    |   movel(pose_trans(ref_frame,p[0.022855, 0.074672, -0.000125, 0.000000, 3.141593, 0.000000]),accel_mss,speed_ms,0,0.001)
    |   movel(pose_trans(ref_frame,p[0.022965, 0.074913, -0.000125, -0.000000, 3.141593, -0.000000]),accel_mss,speed_ms,0,0.001)
    |   movel(pose_trans(ref_frame,p[0.022969, 0.075189, -0.000125, 0.000000, 3.141593, -0.000000]),accel_mss,speed_ms,0,0.001)
    |   movel(pose_trans(ref_frame,p[0.022613, 0.076078, -0.000125, -0.000000, 3.141593, 0.000000]),accel_mss,speed_ms,0,0.001)
    |   movel(pose_trans(ref_frame,p[0.022075, 0.076866, -0.000125, 0.000000, 3.141593, 0.000000]),accel_mss,speed_ms,0,0.001)
    |   movel(pose_trans(ref_frame,p[0.021271, 0.078122, -0.000125, 0.000000, 3.141593, -0.000000]),accel_mss,speed_ms,0,0.001)
    |   movel(pose_trans(ref_frame,p[0.022029, 0.079079, -0.000125, 0.000000, 3.141593, 0.000000]),accel_mss,speed_ms,0,0.001)
    |   movel(pose_trans(ref_frame,p[0.021683, 0.080650, -0.000125, -0.000000, 3.141593, 0.000000]),accel_mss,speed_ms,0,0.001)
    |   movel(pose_trans(ref_frame,p[0.020753, 0.081998, -0.000125, -0.000000, 3.141593, 0.000000]),accel_mss,speed_ms,0,0.001)
    |   movel(pose_trans(ref_frame,p[0.019633, 0.083228, -0.000125, -0.000000, 3.141593, -0.000000]),accel_mss,speed_ms,0,0.001)
    |   movel(pose_trans(ref_frame,p[0.018817, 0.084642, -0.000125, -0.000000, 3.141593, 0.000000]),accel_mss,speed_ms,0,0.001)
    |   movel(pose_trans(ref_frame,p[0.018857, 0.085057, -0.000125, -0.000000, 3.141593, 0.000000]),accel_mss,speed_ms,0,0.001)
    |   movel(pose_trans(ref_frame,p[0.019145, 0.085240, -0.000125, -0.000000, 3.141593, -0.000000]),accel_mss,speed_ms,0,0.001)
    |   movel(pose_trans(ref_frame,p[0.019287, 0.085189, -0.000125, -0.000000, 3.141593, 0.000000]),accel_mss,speed_ms,0,0.001)
    |   movel(pose_trans(ref_frame,p[0.019408, 0.085093, -0.000125, -0.000000, 3.141593, -0.000000]),accel_mss,speed_ms,0,0.001)
    |   movel(pose_trans(ref_frame,p[0.020443, 0.084055, -0.000125, 0.000000, 3.141593, 0.000000]),accel_mss,speed_ms,0,0.001)
    |   movel(pose_trans(ref_frame,p[0.021348, 0.082902, -0.000125, -0.000000, 3.141593, -0.000000]),accel_mss,speed_ms,0,0.001)
    |   movel(pose_trans(ref_frame,p[0.021279, 0.084884, -0.000125, -0.000000, 3.141593, -0.000000]),accel_mss,speed_ms,0,0.001)
    |   movel(pose_trans(ref_frame,p[0.019878, 0.086502, -0.000125, 0.000000, 3.141593, 0.000000]),accel_mss,speed_ms,0,0.001)
    |   movel(pose_trans(ref_frame,p[0.019692, 0.086795, -0.000125, 0.000000, 3.141593, -0.000000]),accel_mss,speed_ms,0,0.001)
    |   movel(pose_trans(ref_frame,p[0.019677, 0.087111, -0.000125, 0.000000, 3.141593, -0.000000]),accel_mss,speed_ms,0,0.001)
    |   movel(pose_trans(ref_frame,p[0.020252, 0.087228, -0.000125, -0.000000, 3.141593, 0.000000]),accel_mss,speed_ms,0,0.001)
    |   movel(pose_trans(ref_frame,p[0.020628, 0.087249, -0.000125, -0.000000, 3.141593, 0.000000]),accel_mss,speed_ms,0,0.001)
    |   movel(pose_trans(ref_frame,p[0.020630, 0.087969, -0.000125, -0.000000, 3.141593, -0.000000]),accel_mss,speed_ms,0,0.001)
    |   movel(pose_trans(ref_frame,p[0.020204, 0.088627, -0.000125, -0.000000, 3.141593, 0.000000]),accel_mss,speed_ms,0,0.001)
    |   movel(pose_trans(ref_frame,p[0.019352, 0.090039, -0.000125, 0.000000, 3.141593, -0.000000]),accel_mss,speed_ms,0,0.001)
    |   movel(pose_trans(ref_frame,p[0.018472, 0.091435, -0.000125, -0.000000, 3.141593, 0.000000]),accel_mss,speed_ms,0,0.001)
    |   movel(pose_trans(ref_frame,p[0.018239, 0.092061, -0.000125, 0.000000, 3.141593, 0.000000]),accel_mss,speed_ms,0,0.001)
    |   movel(pose_trans(ref_frame,p[0.018456, 0.092576, -0.000125, -0.000000, 3.141593, 0.000000]),accel_mss,speed_ms,0,0.001)
    |   movel(pose_trans(ref_frame,p[0.018989, 0.092581, -0.000125, 0.000000, 3.141593, -0.000000]),accel_mss,speed_ms,0,0.001)
    |   movel(pose_trans(ref_frame,p[0.019468, 0.092180, -0.000125, 0.000000, 3.141593, -0.000000]),accel_mss,speed_ms,0,0.001)
    |   movel(pose_trans(ref_frame,p[0.021768, 0.089335, -0.000125, -0.000000, 3.141593, -0.000000]),accel_mss,speed_ms,0,0.001)
    |   movel(pose_trans(ref_frame,p[0.023782, 0.086280, -0.000125, 0.000000, 3.141593, 0.000000]),accel_mss,speed_ms,0,0.001)
    |   movel(pose_trans(ref_frame,p[0.024110, 0.085688, -0.000125, 0.000000, 3.141593, 0.000000]),accel_mss,speed_ms,0,0.001)
    |   movel(pose_trans(ref_frame,p[0.024349, 0.085059, -0.000125, -0.000000, 3.141593, -0.000000]),accel_mss,speed_ms,0,0.001)
    |   movel(pose_trans(ref_frame,p[0.024445, 0.084271, -0.000125, 0.000000, 3.141593, 0.000000]),accel_mss,speed_ms,0,0.001)
    |   movel(pose_trans(ref_frame,p[0.024416, 0.083472, -0.000125, 0.000000, 3.141593, -0.000000]),accel_mss,speed_ms,0,0.001)
    |   movel(pose_trans(ref_frame,p[0.023805, 0.080672, -0.000125, -0.000000, 3.141593, -0.000000]),accel_mss,speed_ms,0,0.001)
    |   movel(pose_trans(ref_frame,p[0.024617, 0.078088, -0.000125, 0.000000, 3.141593, -0.000000]),accel_mss,speed_ms,0,0.001)
    |   movel(pose_trans(ref_frame,p[0.025018, 0.077876, -0.000125, 0.000000, 3.141593, 0.000000]),accel_mss,speed_ms,0,0.001)
    |   movel(pose_trans(ref_frame,p[0.025324, 0.077583, -0.000125, -0.000000, 3.141593, -0.000000]),accel_mss,speed_ms,0,0.001)
    |   movel(pose_trans(ref_frame,p[0.025361, 0.077273, -0.000125, 0.000000, 3.141593, 0.000000]),accel_mss,speed_ms,0,0.001)
    |   movel(pose_trans(ref_frame,p[0.025276, 0.076957, -0.000125, 0.000000, 3.141593, 0.000000]),accel_mss,speed_ms,0,0.001)
    |   movel(pose_trans(ref_frame,p[0.024401, 0.072919, -0.000125, 0.000000, 3.141593, 0.000000]),accel_mss,speed_ms,0,0.001)
    |   movel(pose_trans(ref_frame,p[0.024138, 0.068733, -0.000125, -0.000000, 3.141593, -0.000000]),accel_mss,speed_ms,0,0) # end trace
    |   speed_ms    = 1.000
    |   movel(pose_trans(ref_frame,p[0.024138, 0.068733, 0.005000, -0.000000, 3.141593, -0.000000]),accel_mss,speed_ms,0,0.001)
    |   movel(pose_trans(ref_frame,p[0.024316, 0.065228, 0.005000, -0.000000, 3.141593, -0.000000]),accel_mss,speed_ms,0,0) # end trace
    |   speed_ms    = 0.002
    |   movel(pose_trans(ref_frame,p[0.024316, 0.065228, -0.000125, -0.000000, 3.141593, -0.000000]),accel_mss,speed_ms,0,0) # end trace
    |   speed_ms    = 0.007
    |   movel(pose_trans(ref_frame,p[0.024326, 0.066721, -0.000125, 0.000000, 3.141593, 0.000000]),accel_mss,speed_ms,0,0.001)
    |   movel(pose_trans(ref_frame,p[0.025258, 0.068000, -0.000125, 0.000000, 3.141593, -0.000000]),accel_mss,speed_ms,0,0.001)
    |   movel(pose_trans(ref_frame,p[0.026542, 0.068884, -0.000125, 0.000000, 3.141593, 0.000000]),accel_mss,speed_ms,0,0.001)
    |   movel(pose_trans(ref_frame,p[0.027866, 0.069719, -0.000125, -0.000000, 3.141593, 0.000000]),accel_mss,speed_ms,0,0.001)
    |   movel(pose_trans(ref_frame,p[0.029492, 0.071685, -0.000125, -0.000000, 3.141593, 0.000000]),accel_mss,speed_ms,0,0.001)
    |   movel(pose_trans(ref_frame,p[0.029717, 0.074133, -0.000125, 0.000000, 3.141593, 0.000000]),accel_mss,speed_ms,0,0) # end trace
    |   speed_ms    = 1.000
    |   movel(pose_trans(ref_frame,p[0.029717, 0.074133, 0.005000, 0.000000, 3.141593, -0.000000]),accel_mss,speed_ms,0,0.001)
    |   movel(pose_trans(ref_frame,p[0.025670, 0.079722, 0.005000, -0.000000, 3.141593, -0.000000]),accel_mss,speed_ms,0,0) # end trace
    |   speed_ms    = 0.002
    |   movel(pose_trans(ref_frame,p[0.025670, 0.079722, -0.000125, -0.000000, 3.141593, 0.000000]),accel_mss,speed_ms,0,0) # end trace
    |   speed_ms    = 0.007
    |   movel(pose_trans(ref_frame,p[0.027227, 0.081100, -0.000125, -0.000000, 3.141593, 0.000000]),accel_mss,speed_ms,0,0.001)
    |   movel(pose_trans(ref_frame,p[0.029095, 0.082012, -0.000125, 0.000000, 3.141593, 0.000000]),accel_mss,speed_ms,0,0.001)
    |   movel(pose_trans(ref_frame,p[0.029055, 0.081074, -0.000125, -0.000000, 3.141593, 0.000000]),accel_mss,speed_ms,0,0.001)
    |   movel(pose_trans(ref_frame,p[0.029892, 0.080937, -0.000125, -0.000000, 3.141593, -0.000000]),accel_mss,speed_ms,0,0.001)
    |   movel(pose_trans(ref_frame,p[0.031334, 0.082112, -0.000125, 0.000000, 3.141593, 0.000000]),accel_mss,speed_ms,0,0.001)
    |   movel(pose_trans(ref_frame,p[0.033119, 0.082647, -0.000125, 0.000000, 3.141593, 0.000000]),accel_mss,speed_ms,0,0.001)
    |   movel(pose_trans(ref_frame,p[0.032649, 0.082077, -0.000125, -0.000000, 3.141593, 0.000000]),accel_mss,speed_ms,0,0.001)
    |   movel(pose_trans(ref_frame,p[0.032197, 0.081488, -0.000125, 0.000000, 3.141593, -0.000000]),accel_mss,speed_ms,0,0.001)
    |   movel(pose_trans(ref_frame,p[0.032004, 0.080763, -0.000125, -0.000000, 3.141593, 0.000000]),accel_mss,speed_ms,0,0.001)
    |   movel(pose_trans(ref_frame,p[0.032627, 0.080382, -0.000125, -0.000000, 3.141593, -0.000000]),accel_mss,speed_ms,0,0.001)
    |   movel(pose_trans(ref_frame,p[0.034097, 0.081217, -0.000125, 0.000000, 3.141593, 0.000000]),accel_mss,speed_ms,0,0.001)
    |   movel(pose_trans(ref_frame,p[0.035665, 0.081637, -0.000125, -0.000000, 3.141593, 0.000000]),accel_mss,speed_ms,0,0) # end trace
    |   speed_ms    = 1.000
    |   movel(pose_trans(ref_frame,p[0.035665, 0.081637, 0.005000, -0.000000, 3.141593, -0.000000]),accel_mss,speed_ms,0,0.001)
    |   movel(pose_trans(ref_frame,p[0.040123, 0.075328, 0.005000, -0.000000, 3.141593, -0.000000]),accel_mss,speed_ms,0,0) # end trace
    |   speed_ms    = 0.002
    |   movel(pose_trans(ref_frame,p[0.040123, 0.075328, -0.000125, -0.000000, 3.141593, -0.000000]),accel_mss,speed_ms,0,0) # end trace
    |   speed_ms    = 0.007
    |   movel(pose_trans(ref_frame,p[0.042624, 0.073618, -0.000125, 0.000000, 3.141593, -0.000000]),accel_mss,speed_ms,0,0.001)
    |   movel(pose_trans(ref_frame,p[0.044452, 0.071226, -0.000125, -0.000000, 3.141593, 0.000000]),accel_mss,speed_ms,0,0.001)
    |   movel(pose_trans(ref_frame,p[0.045663, 0.067937, -0.000125, 0.000000, 3.141593, -0.000000]),accel_mss,speed_ms,0,0.001)
    |   movel(pose_trans(ref_frame,p[0.046382, 0.064508, -0.000125, -0.000000, 3.141593, -0.000000]),accel_mss,speed_ms,0,0.001)
    |   movel(pose_trans(ref_frame,p[0.046751, 0.058784, -0.000125, -0.000000, 3.141593, -0.000000]),accel_mss,speed_ms,0,0.001)
    |   movel(pose_trans(ref_frame,p[0.046752, 0.053054, -0.000125, 0.000000, 3.141593, -0.000000]),accel_mss,speed_ms,0,0.001)
    |   movel(pose_trans(ref_frame,p[0.046884, 0.044874, -0.000125, 0.000000, 3.141593, -0.000000]),accel_mss,speed_ms,0,0.001)
    |   movel(pose_trans(ref_frame,p[0.048104, 0.036771, -0.000125, 0.000000, 3.141593, -0.000000]),accel_mss,speed_ms,0,0.001)
    |   movel(pose_trans(ref_frame,p[0.050448, 0.031141, -0.000125, -0.000000, 3.141593, -0.000000]),accel_mss,speed_ms,0,0.001)
    |   movel(pose_trans(ref_frame,p[0.054456, 0.026517, -0.000125, 0.000000, 3.141593, 0.000000]),accel_mss,speed_ms,0,0.001)
    |   movel(pose_trans(ref_frame,p[0.056922, 0.025234, -0.000125, -0.000000, 3.141593, 0.000000]),accel_mss,speed_ms,0,0.001)
    |   movel(pose_trans(ref_frame,p[0.059647, 0.025067, -0.000125, 0.000000, 3.141593, -0.000000]),accel_mss,speed_ms,0,0) # end trace
    |   speed_ms    = 1.000
    |   movel(pose_trans(ref_frame,p[0.059647, 0.025067, 0.005000, 0.000000, 3.141593, 0.000000]),accel_mss,speed_ms,0,0.001)
    |   movel(pose_trans(ref_frame,p[0.043182, 0.008229, 0.005000, -0.000000, 3.141593, 0.000000]),accel_mss,speed_ms,0,0) # end trace
    |   speed_ms    = 0.002
    |   movel(pose_trans(ref_frame,p[0.043182, 0.008229, -0.000125, -0.000000, 3.141593, 0.000000]),accel_mss,speed_ms,0,0) # end trace
    |   speed_ms    = 0.007
    |   movel(pose_trans(ref_frame,p[0.046647, 0.004789, -0.000125, 0.000000, 3.141593, -0.000000]),accel_mss,speed_ms,0,0.001)
    |   movel(pose_trans(ref_frame,p[0.051583, 0.004397, -0.000125, -0.000000, 3.141593, 0.000000]),accel_mss,speed_ms,0,0.001)
    |   movel(pose_trans(ref_frame,p[0.054962, 0.007769, -0.000125, 0.000000, 3.141593, 0.000000]),accel_mss,speed_ms,0,0.001)
    |   movel(pose_trans(ref_frame,p[0.055032, 0.012474, -0.000125, 0.000000, 3.141593, -0.000000]),accel_mss,speed_ms,0,0) # end trace
    |   speed_ms    = 1.000
    |   movel(pose_trans(ref_frame,p[0.055032, 0.012474, 0.005000, 0.000000, 3.141593, 0.000000]),accel_mss,speed_ms,0,0.001)
    |   movel(pose_trans(ref_frame,p[0.021684, 0.038516, 0.005000, -0.000000, 3.141593, -0.000000]),accel_mss,speed_ms,0,0) # end trace
    |   speed_ms    = 0.002
    |   movel(pose_trans(ref_frame,p[0.021684, 0.038516, -0.000125, -0.000000, 3.141593, 0.000000]),accel_mss,speed_ms,0,0) # end trace
    |   speed_ms    = 0.007
    |   movel(pose_trans(ref_frame,p[0.023382, 0.038874, -0.000125, -0.000000, 3.141593, 0.000000]),accel_mss,speed_ms,0,0.001)
    |   movel(pose_trans(ref_frame,p[0.024892, 0.039892, -0.000125, -0.000000, 3.141593, -0.000000]),accel_mss,speed_ms,0,0.001)
    |   movel(pose_trans(ref_frame,p[0.026323, 0.041126, -0.000125, 0.000000, 3.141593, -0.000000]),accel_mss,speed_ms,0,0.001)
    |   movel(pose_trans(ref_frame,p[0.027311, 0.042675, -0.000125, -0.000000, 3.141593, -0.000000]),accel_mss,speed_ms,0,0.001)
    |   movel(pose_trans(ref_frame,p[0.027536, 0.044188, -0.000125, 0.000000, 3.141593, -0.000000]),accel_mss,speed_ms,0,0.001)
    |   movel(pose_trans(ref_frame,p[0.027568, 0.045740, -0.000125, 0.000000, 3.141593, -0.000000]),accel_mss,speed_ms,0,0.001)
    |   movel(pose_trans(ref_frame,p[0.028234, 0.047523, -0.000125, -0.000000, 3.141593, 0.000000]),accel_mss,speed_ms,0,0.001)
    |   movel(pose_trans(ref_frame,p[0.029388, 0.049022, -0.000125, 0.000000, 3.141593, -0.000000]),accel_mss,speed_ms,0,0.001)
    |   movel(pose_trans(ref_frame,p[0.030515, 0.051231, -0.000125, 0.000000, 3.141593, -0.000000]),accel_mss,speed_ms,0,0.001)
    |   movel(pose_trans(ref_frame,p[0.030773, 0.053692, -0.000125, -0.000000, 3.141593, -0.000000]),accel_mss,speed_ms,0,0) # end trace
    |   speed_ms    = 1.000
    |   movel(pose_trans(ref_frame,p[0.030773, 0.053692, 0.005000, -0.000000, 3.141593, -0.000000]),accel_mss,speed_ms,0,0.001)
    |   movel(pose_trans(ref_frame,p[0.028356, 0.053295, 0.005000, 0.000000, 3.141593, 0.000000]),accel_mss,speed_ms,0,0) # end trace
    |   speed_ms    = 0.002
    |   movel(pose_trans(ref_frame,p[0.028356, 0.053295, -0.000125, 0.000000, 3.141593, 0.000000]),accel_mss,speed_ms,0,0) # end trace
    |   speed_ms    = 0.007
    |   movel(pose_trans(ref_frame,p[0.027850, 0.051369, -0.000125, -0.000000, 3.141593, -0.000000]),accel_mss,speed_ms,0,0.001)
    |   movel(pose_trans(ref_frame,p[0.026989, 0.049584, -0.000125, 0.000000, 3.141593, -0.000000]),accel_mss,speed_ms,0,0.001)
    |   movel(pose_trans(ref_frame,p[0.026294, 0.047720, -0.000125, -0.000000, 3.141593, -0.000000]),accel_mss,speed_ms,0,0.001)
    |   movel(pose_trans(ref_frame,p[0.025945, 0.045753, -0.000125, -0.000000, 3.141593, 0.000000]),accel_mss,speed_ms,0,0.001)
    |   movel(pose_trans(ref_frame,p[0.025882, 0.044781, -0.000125, -0.000000, 3.141593, 0.000000]),accel_mss,speed_ms,0,0.001)
    |   movel(pose_trans(ref_frame,p[0.025835, 0.043807, -0.000125, 0.000000, 3.141593, -0.000000]),accel_mss,speed_ms,0,0.001)
    |   movel(pose_trans(ref_frame,p[0.025824, 0.043717, -0.000125, 0.000000, 3.141593, -0.000000]),accel_mss,speed_ms,0,0.001)
    |   movel(pose_trans(ref_frame,p[0.025784, 0.043638, -0.000125, 0.000000, 3.141593, -0.000000]),accel_mss,speed_ms,0,0.001)
    |   movel(pose_trans(ref_frame,p[0.025697, 0.043586, -0.000125, 0.000000, 3.141593, -0.000000]),accel_mss,speed_ms,0,0.001)
    |   movel(pose_trans(ref_frame,p[0.025593, 0.043571, -0.000125, 0.000000, 3.141593, -0.000000]),accel_mss,speed_ms,0,0.001)
    |   movel(pose_trans(ref_frame,p[0.024730, 0.043675, -0.000125, 0.000000, 3.141593, -0.000000]),accel_mss,speed_ms,0,0.001)
    |   movel(pose_trans(ref_frame,p[0.023962, 0.044084, -0.000125, 0.000000, 3.141593, 0.000000]),accel_mss,speed_ms,0,0.001)
    |   movel(pose_trans(ref_frame,p[0.024473, 0.043044, -0.000125, 0.000000, 3.141593, -0.000000]),accel_mss,speed_ms,0,0.001)
    |   movel(pose_trans(ref_frame,p[0.025091, 0.042066, -0.000125, 0.000000, 3.141593, 0.000000]),accel_mss,speed_ms,0,0.001)
    |   movel(pose_trans(ref_frame,p[0.023980, 0.040968, -0.000125, 0.000000, 3.141593, -0.000000]),accel_mss,speed_ms,0,0.001)
    |   movel(pose_trans(ref_frame,p[0.022648, 0.040143, -0.000125, -0.000000, 3.141593, -0.000000]),accel_mss,speed_ms,0,0.001)
    |   movel(pose_trans(ref_frame,p[0.022358, 0.040021, -0.000125, -0.000000, 3.141593, -0.000000]),accel_mss,speed_ms,0,0.001)
    |   movel(pose_trans(ref_frame,p[0.022053, 0.039950, -0.000125, -0.000000, 3.141593, -0.000000]),accel_mss,speed_ms,0,0.001)
    |   movel(pose_trans(ref_frame,p[0.020963, 0.040215, -0.000125, -0.000000, 3.141593, -0.000000]),accel_mss,speed_ms,0,0.001)
    |   movel(pose_trans(ref_frame,p[0.020018, 0.040782, -0.000125, 0.000000, 3.141593, 0.000000]),accel_mss,speed_ms,0,0.001)
    |   movel(pose_trans(ref_frame,p[0.019840, 0.040545, -0.000125, 0.000000, 3.141593, -0.000000]),accel_mss,speed_ms,0,0.001)
    |   movel(pose_trans(ref_frame,p[0.020104, 0.040193, -0.000125, 0.000000, 3.141593, -0.000000]),accel_mss,speed_ms,0,0.001)
    |   movel(pose_trans(ref_frame,p[0.020326, 0.039832, -0.000125, -0.000000, 3.141593, -0.000000]),accel_mss,speed_ms,0,0.001)
    |   movel(pose_trans(ref_frame,p[0.020579, 0.039493, -0.000125, 0.000000, 3.141593, 0.000000]),accel_mss,speed_ms,0,0.001)
    |   movel(pose_trans(ref_frame,p[0.021024, 0.039057, -0.000125, 0.000000, 3.141593, -0.000000]),accel_mss,speed_ms,0,0.001)
    |   movel(pose_trans(ref_frame,p[0.021049, 0.039080, -0.000125, 0.000000, 3.141593, -0.000000]),accel_mss,speed_ms,0,0) # end trace
    |   speed_ms    = 1.000
    |   movel(pose_trans(ref_frame,p[0.021049, 0.039080, 0.005000, 0.000000, 3.141593, 0.000000]),accel_mss,speed_ms,0,0.001)
    |   movel(pose_trans(ref_frame,p[0.018458, 0.040911, 0.005000, 0.000000, 3.141593, -0.000000]),accel_mss,speed_ms,0,0) # end trace
    |   speed_ms    = 0.002
    |   movel(pose_trans(ref_frame,p[0.018458, 0.040911, -0.000125, 0.000000, 3.141593, -0.000000]),accel_mss,speed_ms,0,0) # end trace
    |   speed_ms    = 0.007
    |   movel(pose_trans(ref_frame,p[0.018326, 0.037997, -0.000125, 0.000000, 3.141593, 0.000000]),accel_mss,speed_ms,0,0.001)
    |   movel(pose_trans(ref_frame,p[0.019055, 0.035242, -0.000125, 0.000000, 3.141593, -0.000000]),accel_mss,speed_ms,0,0.001)
    |   movel(pose_trans(ref_frame,p[0.019471, 0.037804, -0.000125, 0.000000, 3.141593, -0.000000]),accel_mss,speed_ms,0,0.001)
    |   movel(pose_trans(ref_frame,p[0.020491, 0.035398, -0.000125, 0.000000, 3.141593, -0.000000]),accel_mss,speed_ms,0,0.001)
    |   movel(pose_trans(ref_frame,p[0.022615, 0.034140, -0.000125, 0.000000, 3.141593, -0.000000]),accel_mss,speed_ms,0,0.001)
    |   movel(pose_trans(ref_frame,p[0.021937, 0.035325, -0.000125, -0.000000, 3.141593, 0.000000]),accel_mss,speed_ms,0,0.001)
    |   movel(pose_trans(ref_frame,p[0.021623, 0.036608, -0.000125, 0.000000, 3.141593, -0.000000]),accel_mss,speed_ms,0,0.001)
    |   movel(pose_trans(ref_frame,p[0.023117, 0.035906, -0.000125, 0.000000, 3.141593, -0.000000]),accel_mss,speed_ms,0,0.001)
    |   movel(pose_trans(ref_frame,p[0.024737, 0.035089, -0.000125, -0.000000, 3.141593, -0.000000]),accel_mss,speed_ms,0,0.001)
    |   movel(pose_trans(ref_frame,p[0.024951, 0.035728, -0.000125, -0.000000, 3.141593, -0.000000]),accel_mss,speed_ms,0,0.001)
    |   movel(pose_trans(ref_frame,p[0.025019, 0.036399, -0.000125, -0.000000, 3.141593, -0.000000]),accel_mss,speed_ms,0,0.001)
    |   movel(pose_trans(ref_frame,p[0.026135, 0.036108, -0.000125, -0.000000, 3.141593, -0.000000]),accel_mss,speed_ms,0,0.001)
    |   movel(pose_trans(ref_frame,p[0.027105, 0.035487, -0.000125, -0.000000, 3.141593, 0.000000]),accel_mss,speed_ms,0,0.001)
    |   movel(pose_trans(ref_frame,p[0.027535, 0.035653, -0.000125, 0.000000, 3.141593, -0.000000]),accel_mss,speed_ms,0,0.001)
    |   movel(pose_trans(ref_frame,p[0.027831, 0.037320, -0.000125, 0.000000, 3.141593, -0.000000]),accel_mss,speed_ms,0,0.001)
    |   movel(pose_trans(ref_frame,p[0.027963, 0.038300, -0.000125, -0.000000, 3.141593, 0.000000]),accel_mss,speed_ms,0,0.001)
    |   movel(pose_trans(ref_frame,p[0.027938, 0.039314, -0.000125, 0.000000, 3.141593, -0.000000]),accel_mss,speed_ms,0,0.001)
    |   movel(pose_trans(ref_frame,p[0.028745, 0.038587, -0.000125, -0.000000, 3.141593, -0.000000]),accel_mss,speed_ms,0,0.001)
    |   movel(pose_trans(ref_frame,p[0.029553, 0.037860, -0.000125, 0.000000, 3.141593, -0.000000]),accel_mss,speed_ms,0,0.001)
    |   movel(pose_trans(ref_frame,p[0.029813, 0.040047, -0.000125, -0.000000, 3.141593, 0.000000]),accel_mss,speed_ms,0,0.001)
    |   movel(pose_trans(ref_frame,p[0.029469, 0.042222, -0.000125, 0.000000, 3.141593, -0.000000]),accel_mss,speed_ms,0,0.001)
    |   movel(pose_trans(ref_frame,p[0.029405, 0.042550, -0.000125, 0.000000, 3.141593, -0.000000]),accel_mss,speed_ms,0,0.001)
    |   movel(pose_trans(ref_frame,p[0.029469, 0.042855, -0.000125, 0.000000, 3.141593, -0.000000]),accel_mss,speed_ms,0,0.001)
    |   movel(pose_trans(ref_frame,p[0.029623, 0.043004, -0.000125, 0.000000, 3.141593, 0.000000]),accel_mss,speed_ms,0,0.001)
    |   movel(pose_trans(ref_frame,p[0.029817, 0.043105, -0.000125, -0.000000, 3.141593, -0.000000]),accel_mss,speed_ms,0,0.001)
    |   movel(pose_trans(ref_frame,p[0.030735, 0.043743, -0.000125, 0.000000, 3.141593, 0.000000]),accel_mss,speed_ms,0,0.001)
    |   movel(pose_trans(ref_frame,p[0.032075, 0.043686, -0.000125, -0.000000, 3.141593, -0.000000]),accel_mss,speed_ms,0,0.001)
    |   movel(pose_trans(ref_frame,p[0.031242, 0.044530, -0.000125, 0.000000, 3.141593, -0.000000]),accel_mss,speed_ms,0,0.001)
    |   movel(pose_trans(ref_frame,p[0.030296, 0.045244, -0.000125, 0.000000, 3.141593, 0.000000]),accel_mss,speed_ms,0,0.001)
    |   movel(pose_trans(ref_frame,p[0.032373, 0.047290, -0.000125, -0.000000, 3.141593, 0.000000]),accel_mss,speed_ms,0,0.001)
    |   movel(pose_trans(ref_frame,p[0.033820, 0.049803, -0.000125, 0.000000, 3.141593, 0.000000]),accel_mss,speed_ms,0,0.001)
    |   movel(pose_trans(ref_frame,p[0.032727, 0.049289, -0.000125, 0.000000, 3.141593, -0.000000]),accel_mss,speed_ms,0,0.001)
    |   movel(pose_trans(ref_frame,p[0.031535, 0.049066, -0.000125, -0.000000, 3.141593, 0.000000]),accel_mss,speed_ms,0,0.001)
    |   movel(pose_trans(ref_frame,p[0.032744, 0.050356, -0.000125, 0.000000, 3.141593, -0.000000]),accel_mss,speed_ms,0,0.001)
    |   movel(pose_trans(ref_frame,p[0.033365, 0.052011, -0.000125, -0.000000, 3.141593, -0.000000]),accel_mss,speed_ms,0,0) # end trace
    |   speed_ms    = 1.000
    |   movel(pose_trans(ref_frame,p[0.033365, 0.052011, 0.005000, -0.000000, 3.141593, 0.000000]),accel_mss,speed_ms,0,0.001)
    |   movel(pose_trans(ref_frame,p[0.026398, 0.054187, 0.005000, 0.000000, 3.141593, -0.000000]),accel_mss,speed_ms,0,0) # end trace
    |   speed_ms    = 0.002
    |   movel(pose_trans(ref_frame,p[0.026398, 0.054187, -0.000125, 0.000000, 3.141593, -0.000000]),accel_mss,speed_ms,0,0) # end trace
    |   speed_ms    = 0.007
    |   movel(pose_trans(ref_frame,p[0.027548, 0.056488, -0.000125, -0.000000, 3.141593, -0.000000]),accel_mss,speed_ms,0,0.001)
    |   movel(pose_trans(ref_frame,p[0.028692, 0.058780, -0.000125, -0.000000, 3.141593, -0.000000]),accel_mss,speed_ms,0,0.001)
    |   movel(pose_trans(ref_frame,p[0.028756, 0.058934, -0.000125, -0.000000, 3.141593, -0.000000]),accel_mss,speed_ms,0,0.001)
    |   movel(pose_trans(ref_frame,p[0.028788, 0.059094, -0.000125, -0.000000, 3.141593, 0.000000]),accel_mss,speed_ms,0,0.001)
    |   movel(pose_trans(ref_frame,p[0.028750, 0.059295, -0.000125, -0.000000, 3.141593, 0.000000]),accel_mss,speed_ms,0,0.001)
    |   movel(pose_trans(ref_frame,p[0.028674, 0.059488, -0.000125, -0.000000, 3.141593, -0.000000]),accel_mss,speed_ms,0,0.001)
    |   movel(pose_trans(ref_frame,p[0.028528, 0.059997, -0.000125, 0.000000, 3.141593, 0.000000]),accel_mss,speed_ms,0,0.001)
    |   movel(pose_trans(ref_frame,p[0.028496, 0.060526, -0.000125, 0.000000, 3.141593, 0.000000]),accel_mss,speed_ms,0,0) # end trace
    |   speed_ms    = 1.000
    |   movel(pose_trans(ref_frame,p[0.028496, 0.060526, 0.005000, 0.000000, 3.141593, 0.000000]),accel_mss,speed_ms,0,0.001)
    |   movel(pose_trans(ref_frame,p[0.027012, 0.061022, 0.005000, -0.000000, 3.141593, 0.000000]),accel_mss,speed_ms,0,0) # end trace
    |   speed_ms    = 0.002
    |   movel(pose_trans(ref_frame,p[0.027012, 0.061022, -0.000125, 0.000000, 3.141593, -0.000000]),accel_mss,speed_ms,0,0) # end trace
    |   speed_ms    = 0.007
    |   movel(pose_trans(ref_frame,p[0.026991, 0.061048, -0.000125, 0.000000, 3.141593, 0.000000]),accel_mss,speed_ms,0,0.001)
    |   movel(pose_trans(ref_frame,p[0.029212, 0.062985, -0.000125, 0.000000, 3.141593, -0.000000]),accel_mss,speed_ms,0,0.001)
    |   movel(pose_trans(ref_frame,p[0.031074, 0.064473, -0.000125, 0.000000, 3.141593, -0.000000]),accel_mss,speed_ms,0,0.001)
    |   movel(pose_trans(ref_frame,p[0.032138, 0.066587, -0.000125, -0.000000, 3.141593, -0.000000]),accel_mss,speed_ms,0,0.001)
    |   movel(pose_trans(ref_frame,p[0.032261, 0.067208, -0.000125, 0.000000, 3.141593, -0.000000]),accel_mss,speed_ms,0,0.001)
    |   movel(pose_trans(ref_frame,p[0.032292, 0.067836, -0.000125, -0.000000, 3.141593, -0.000000]),accel_mss,speed_ms,0,0.001)
    |   movel(pose_trans(ref_frame,p[0.032271, 0.068503, -0.000125, 0.000000, 3.141593, -0.000000]),accel_mss,speed_ms,0,0.001)
    |   movel(pose_trans(ref_frame,p[0.031727, 0.068972, -0.000125, 0.000000, 3.141593, 0.000000]),accel_mss,speed_ms,0,0.001)
    |   movel(pose_trans(ref_frame,p[0.031486, 0.068682, -0.000125, -0.000000, 3.141593, -0.000000]),accel_mss,speed_ms,0,0.001)
    |   movel(pose_trans(ref_frame,p[0.031083, 0.068111, -0.000125, 0.000000, 3.141593, -0.000000]),accel_mss,speed_ms,0,0) # end trace
    |   speed_ms    = 1.000
    |   movel(pose_trans(ref_frame,p[0.031083, 0.068111, 0.005000, 0.000000, 3.141593, 0.000000]),accel_mss,speed_ms,0,0.001)
    |   movel(pose_trans(ref_frame,p[0.030129, 0.063246, 0.005000, 0.000000, 3.141593, 0.000000]),accel_mss,speed_ms,0,0) # end trace
    |   speed_ms    = 0.002
    |   movel(pose_trans(ref_frame,p[0.030129, 0.063246, -0.000125, 0.000000, 3.141593, 0.000000]),accel_mss,speed_ms,0,0) # end trace
    |   speed_ms    = 0.007
    |   movel(pose_trans(ref_frame,p[0.031155, 0.062092, -0.000125, 0.000000, 3.141593, 0.000000]),accel_mss,speed_ms,0,0.001)
    |   movel(pose_trans(ref_frame,p[0.032501, 0.061271, -0.000125, -0.000000, 3.141593, -0.000000]),accel_mss,speed_ms,0,0.001)
    |   movel(pose_trans(ref_frame,p[0.032739, 0.061130, -0.000125, -0.000000, 3.141593, -0.000000]),accel_mss,speed_ms,0,0.001)
    |   movel(pose_trans(ref_frame,p[0.032899, 0.060921, -0.000125, 0.000000, 3.141593, -0.000000]),accel_mss,speed_ms,0,0.001)
    |   movel(pose_trans(ref_frame,p[0.032918, 0.060742, -0.000125, 0.000000, 3.141593, 0.000000]),accel_mss,speed_ms,0,0.001)
    |   movel(pose_trans(ref_frame,p[0.032886, 0.060560, -0.000125, -0.000000, 3.141593, 0.000000]),accel_mss,speed_ms,0,0.001)
    |   movel(pose_trans(ref_frame,p[0.032508, 0.058699, -0.000125, 0.000000, 3.141593, -0.000000]),accel_mss,speed_ms,0,0.001)
    |   movel(pose_trans(ref_frame,p[0.032479, 0.058579, -0.000125, 0.000000, 3.141593, -0.000000]),accel_mss,speed_ms,0,0.001)
    |   movel(pose_trans(ref_frame,p[0.032428, 0.058469, -0.000125, -0.000000, 3.141593, -0.000000]),accel_mss,speed_ms,0,0.001)
    |   movel(pose_trans(ref_frame,p[0.032326, 0.058368, -0.000125, 0.000000, 3.141593, -0.000000]),accel_mss,speed_ms,0,0.001)
    |   movel(pose_trans(ref_frame,p[0.032204, 0.058287, -0.000125, 0.000000, 3.141593, -0.000000]),accel_mss,speed_ms,0,0.001)
    |   movel(pose_trans(ref_frame,p[0.031471, 0.057388, -0.000125, -0.000000, 3.141593, -0.000000]),accel_mss,speed_ms,0,0.001)
    |   movel(pose_trans(ref_frame,p[0.031142, 0.056224, -0.000125, 0.000000, 3.141593, 0.000000]),accel_mss,speed_ms,0,0) # end trace
    |   speed_ms    = 1.000
    |   movel(pose_trans(ref_frame,p[0.031142, 0.056224, 0.005000, 0.000000, 3.141593, 0.000000]),accel_mss,speed_ms,0,0.001)
    |   movel(pose_trans(ref_frame,p[0.029444, 0.062095, 0.005000, 0.000000, 3.141593, 0.000000]),accel_mss,speed_ms,0,0) # end trace
    |   speed_ms    = 0.002
    |   movel(pose_trans(ref_frame,p[0.029444, 0.062095, -0.000125, 0.000000, 3.141593, 0.000000]),accel_mss,speed_ms,0,0) # end trace
    |   speed_ms    = 0.007
    |   movel(pose_trans(ref_frame,p[0.030414, 0.061365, -0.000125, 0.000000, 3.141593, 0.000000]),accel_mss,speed_ms,0,0.001)
    |   movel(pose_trans(ref_frame,p[0.030979, 0.060193, -0.000125, 0.000000, 3.141593, -0.000000]),accel_mss,speed_ms,0,0.001)
    |   movel(pose_trans(ref_frame,p[0.031017, 0.060081, -0.000125, 0.000000, 3.141593, 0.000000]),accel_mss,speed_ms,0,0.001)
    |   movel(pose_trans(ref_frame,p[0.031035, 0.059966, -0.000125, -0.000000, 3.141593, -0.000000]),accel_mss,speed_ms,0,0.001)
    |   movel(pose_trans(ref_frame,p[0.031003, 0.059792, -0.000125, -0.000000, 3.141593, -0.000000]),accel_mss,speed_ms,0,0.001)
    |   movel(pose_trans(ref_frame,p[0.030930, 0.059628, -0.000125, -0.000000, 3.141593, -0.000000]),accel_mss,speed_ms,0,0.001)
    |   movel(pose_trans(ref_frame,p[0.030115, 0.057804, -0.000125, -0.000000, 3.141593, -0.000000]),accel_mss,speed_ms,0,0.001)
    |   movel(pose_trans(ref_frame,p[0.029454, 0.055918, -0.000125, 0.000000, 3.141593, -0.000000]),accel_mss,speed_ms,0,0) # end trace
    |   speed_ms    = 1.000
    |   movel(pose_trans(ref_frame,p[0.029454, 0.055918, 0.005000, 0.000000, 3.141593, 0.000000]),accel_mss,speed_ms,0,0.001)
    |   movel(pose_trans(ref_frame,p[0.023891, 0.052575, 0.005000, 0.000000, 3.141593, -0.000000]),accel_mss,speed_ms,0,0) # end trace
    |   speed_ms    = 0.002
    |   movel(pose_trans(ref_frame,p[0.023891, 0.052575, -0.000125, 0.000000, 3.141593, 0.000000]),accel_mss,speed_ms,0,0) # end trace
    |   speed_ms    = 0.007
    |   movel(pose_trans(ref_frame,p[0.024280, 0.054141, -0.000125, -0.000000, 3.141593, 0.000000]),accel_mss,speed_ms,0,0.001)
    |   movel(pose_trans(ref_frame,p[0.025195, 0.055469, -0.000125, -0.000000, 3.141593, 0.000000]),accel_mss,speed_ms,0,0) # end trace
    |   speed_ms    = 1.000
    |   movel(pose_trans(ref_frame,p[0.025195, 0.055469, 0.005000, -0.000000, 3.141593, 0.000000]),accel_mss,speed_ms,0,0.001)
    |   movel(pose_trans(ref_frame,p[0.022695, 0.052030, 0.005000, -0.000000, 3.141593, -0.000000]),accel_mss,speed_ms,0,0) # end trace
    |   speed_ms    = 0.002
    |   movel(pose_trans(ref_frame,p[0.022695, 0.052030, -0.000125, 0.000000, 3.141593, 0.000000]),accel_mss,speed_ms,0,0) # end trace
    |   speed_ms    = 0.007
    |   movel(pose_trans(ref_frame,p[0.022851, 0.052621, -0.000125, 0.000000, 3.141593, -0.000000]),accel_mss,speed_ms,0,0.001)
    |   movel(pose_trans(ref_frame,p[0.023052, 0.053213, -0.000125, -0.000000, 3.141593, -0.000000]),accel_mss,speed_ms,0,0.001)
    |   movel(pose_trans(ref_frame,p[0.023514, 0.053884, -0.000125, -0.000000, 3.141593, -0.000000]),accel_mss,speed_ms,0,0.001)
    |   movel(pose_trans(ref_frame,p[0.024073, 0.054474, -0.000125, 0.000000, 3.141593, -0.000000]),accel_mss,speed_ms,0,0.001)
    |   movel(pose_trans(ref_frame,p[0.024746, 0.055091, -0.000125, -0.000000, 3.141593, -0.000000]),accel_mss,speed_ms,0,0.001)
    |   movel(pose_trans(ref_frame,p[0.025419, 0.055710, -0.000125, -0.000000, 3.141593, -0.000000]),accel_mss,speed_ms,0,0.001)
    |   movel(pose_trans(ref_frame,p[0.026946, 0.058100, -0.000125, 0.000000, 3.141593, -0.000000]),accel_mss,speed_ms,0,0.001)
    |   movel(pose_trans(ref_frame,p[0.027857, 0.060847, -0.000125, -0.000000, 3.141593, 0.000000]),accel_mss,speed_ms,0,0) # end trace
    |   speed_ms    = 1.000
    |   movel(pose_trans(ref_frame,p[0.027857, 0.060847, 0.005000, -0.000000, 3.141593, 0.000000]),accel_mss,speed_ms,0,0.001)
    |   movel(pose_trans(ref_frame,p[0.025348, 0.062306, 0.005000, 0.000000, 3.141593, -0.000000]),accel_mss,speed_ms,0,0) # end trace
    |   speed_ms    = 0.002
    |   movel(pose_trans(ref_frame,p[0.025348, 0.062306, -0.000125, 0.000000, 3.141593, 0.000000]),accel_mss,speed_ms,0,0) # end trace
    |   speed_ms    = 0.007
    |   movel(pose_trans(ref_frame,p[0.025394, 0.063147, -0.000125, -0.000000, 3.141593, -0.000000]),accel_mss,speed_ms,0,0.001)
    |   movel(pose_trans(ref_frame,p[0.025440, 0.063989, -0.000125, -0.000000, 3.141593, -0.000000]),accel_mss,speed_ms,0,0.001)
    |   movel(pose_trans(ref_frame,p[0.025482, 0.064473, -0.000125, -0.000000, 3.141593, -0.000000]),accel_mss,speed_ms,0,0.001)
    |   movel(pose_trans(ref_frame,p[0.025615, 0.064934, -0.000125, 0.000000, 3.141593, 0.000000]),accel_mss,speed_ms,0,0.001)
    |   movel(pose_trans(ref_frame,p[0.026265, 0.065631, -0.000125, 0.000000, 3.141593, 0.000000]),accel_mss,speed_ms,0,0.001)
    |   movel(pose_trans(ref_frame,p[0.027136, 0.066124, -0.000125, -0.000000, 3.141593, 0.000000]),accel_mss,speed_ms,0,0.001)
    |   movel(pose_trans(ref_frame,p[0.028038, 0.066767, -0.000125, 0.000000, 3.141593, 0.000000]),accel_mss,speed_ms,0,0.001)
    |   movel(pose_trans(ref_frame,p[0.028798, 0.067574, -0.000125, 0.000000, 3.141593, 0.000000]),accel_mss,speed_ms,0,0.001)
    |   movel(pose_trans(ref_frame,p[0.029298, 0.068532, -0.000125, -0.000000, 3.141593, 0.000000]),accel_mss,speed_ms,0,0.001)
    |   movel(pose_trans(ref_frame,p[0.029776, 0.069485, -0.000125, 0.000000, 3.141593, -0.000000]),accel_mss,speed_ms,0,0.001)
    |   movel(pose_trans(ref_frame,p[0.029875, 0.069476, -0.000125, 0.000000, 3.141593, 0.000000]),accel_mss,speed_ms,0,0.001)
    |   movel(pose_trans(ref_frame,p[0.030391, 0.068153, -0.000125, 0.000000, 3.141593, -0.000000]),accel_mss,speed_ms,0,0.001)
    |   movel(pose_trans(ref_frame,p[0.030401, 0.067412, -0.000125, -0.000000, 3.141593, 0.000000]),accel_mss,speed_ms,0,0.001)
    |   movel(pose_trans(ref_frame,p[0.030174, 0.066707, -0.000125, -0.000000, 3.141593, -0.000000]),accel_mss,speed_ms,0,0.001)
    |   movel(pose_trans(ref_frame,p[0.027555, 0.064758, -0.000125, 0.000000, 3.141593, -0.000000]),accel_mss,speed_ms,0,0.001)
    |   movel(pose_trans(ref_frame,p[0.026457, 0.063176, -0.000125, 0.000000, 3.141593, 0.000000]),accel_mss,speed_ms,0,0) # end trace
    |   speed_ms    = 1.000
    |   movel(pose_trans(ref_frame,p[0.026457, 0.063176, 0.005000, 0.000000, 3.141593, 0.000000]),accel_mss,speed_ms,0,0.001)
    |   movel(pose_trans(ref_frame,p[0.022436, 0.059610, 0.005000, -0.000000, 3.141593, 0.000000]),accel_mss,speed_ms,0,0) # end trace
    |   speed_ms    = 0.002
    |   movel(pose_trans(ref_frame,p[0.022436, 0.059610, -0.000125, -0.000000, 3.141593, -0.000000]),accel_mss,speed_ms,0,0) # end trace
    |   speed_ms    = 0.007
    |   movel(pose_trans(ref_frame,p[0.022442, 0.059575, -0.000125, 0.000000, 3.141593, 0.000000]),accel_mss,speed_ms,0,0.001)
    |   movel(pose_trans(ref_frame,p[0.022448, 0.059540, -0.000125, -0.000000, 3.141593, 0.000000]),accel_mss,speed_ms,0,0.001)
    |   movel(pose_trans(ref_frame,p[0.022444, 0.057910, -0.000125, 0.000000, 3.141593, -0.000000]),accel_mss,speed_ms,0,0.001)
    |   movel(pose_trans(ref_frame,p[0.021817, 0.056442, -0.000125, -0.000000, 3.141593, -0.000000]),accel_mss,speed_ms,0,0.001)
    |   movel(pose_trans(ref_frame,p[0.021542, 0.056125, -0.000125, -0.000000, 3.141593, 0.000000]),accel_mss,speed_ms,0,0.001)
    |   movel(pose_trans(ref_frame,p[0.021216, 0.055865, -0.000125, -0.000000, 3.141593, 0.000000]),accel_mss,speed_ms,0,0.001)
    |   movel(pose_trans(ref_frame,p[0.020322, 0.055587, -0.000125, 0.000000, 3.141593, 0.000000]),accel_mss,speed_ms,0,0.001)
    |   movel(pose_trans(ref_frame,p[0.019400, 0.055703, -0.000125, 0.000000, 3.141593, -0.000000]),accel_mss,speed_ms,0,0.001)
    |   movel(pose_trans(ref_frame,p[0.020842, 0.055251, -0.000125, 0.000000, 3.141593, -0.000000]),accel_mss,speed_ms,0,0.001)
    |   movel(pose_trans(ref_frame,p[0.022225, 0.055388, -0.000125, 0.000000, 3.141593, 0.000000]),accel_mss,speed_ms,0,0.001)
    |   movel(pose_trans(ref_frame,p[0.022791, 0.055888, -0.000125, -0.000000, 3.141593, 0.000000]),accel_mss,speed_ms,0,0.001)
    |   movel(pose_trans(ref_frame,p[0.023168, 0.056558, -0.000125, 0.000000, 3.141593, 0.000000]),accel_mss,speed_ms,0,0.001)
    |   movel(pose_trans(ref_frame,p[0.023462, 0.057628, -0.000125, 0.000000, 3.141593, -0.000000]),accel_mss,speed_ms,0,0.001)
    |   movel(pose_trans(ref_frame,p[0.023477, 0.058737, -0.000125, 0.000000, 3.141593, 0.000000]),accel_mss,speed_ms,0,0) # end trace
    |   speed_ms    = 1.000
    |   movel(pose_trans(ref_frame,p[0.023477, 0.058737, 0.005000, 0.000000, 3.141593, 0.000000]),accel_mss,speed_ms,0,0.001)
    |   movel(pose_trans(ref_frame,p[0.021306, 0.057911, 0.005000, 0.000000, 3.141593, -0.000000]),accel_mss,speed_ms,0,0) # end trace
    |   speed_ms    = 0.002
    |   movel(pose_trans(ref_frame,p[0.021306, 0.057911, -0.000125, 0.000000, 3.141593, 0.000000]),accel_mss,speed_ms,0,0) # end trace
    |   speed_ms    = 0.007
    |   movel(pose_trans(ref_frame,p[0.021283, 0.057777, -0.000125, -0.000000, 3.141593, 0.000000]),accel_mss,speed_ms,0,0.001)
    |   movel(pose_trans(ref_frame,p[0.021293, 0.057646, -0.000125, 0.000000, 3.141593, 0.000000]),accel_mss,speed_ms,0,0.001)
    |   movel(pose_trans(ref_frame,p[0.021376, 0.057539, -0.000125, -0.000000, 3.141593, 0.000000]),accel_mss,speed_ms,0,0.001)
    |   movel(pose_trans(ref_frame,p[0.021501, 0.057527, -0.000125, 0.000000, 3.141593, -0.000000]),accel_mss,speed_ms,0,0.001)
    |   movel(pose_trans(ref_frame,p[0.021552, 0.057562, -0.000125, 0.000000, 3.141593, 0.000000]),accel_mss,speed_ms,0,0.001)
    |   movel(pose_trans(ref_frame,p[0.021593, 0.057610, -0.000125, 0.000000, 3.141593, 0.000000]),accel_mss,speed_ms,0,0.001)
    |   movel(pose_trans(ref_frame,p[0.021664, 0.057728, -0.000125, -0.000000, 3.141593, 0.000000]),accel_mss,speed_ms,0,0.001)
    |   movel(pose_trans(ref_frame,p[0.021697, 0.057860, -0.000125, 0.000000, 3.141593, -0.000000]),accel_mss,speed_ms,0,0.001)
    |   movel(pose_trans(ref_frame,p[0.021664, 0.057994, -0.000125, 0.000000, 3.141593, -0.000000]),accel_mss,speed_ms,0,0.001)
    |   movel(pose_trans(ref_frame,p[0.021564, 0.058078, -0.000125, 0.000000, 3.141593, -0.000000]),accel_mss,speed_ms,0,0.001)
    |   movel(pose_trans(ref_frame,p[0.021431, 0.058056, -0.000125, 0.000000, 3.141593, 0.000000]),accel_mss,speed_ms,0,0.001)
    |   movel(pose_trans(ref_frame,p[0.021382, 0.057938, -0.000125, -0.000000, 3.141593, 0.000000]),accel_mss,speed_ms,0,0) # end trace
    |   speed_ms    = 1.000
    |   movel(pose_trans(ref_frame,p[0.021382, 0.057938, 0.005000, -0.000000, 3.141593, 0.000000]),accel_mss,speed_ms,0,0.001)
    |   movel(pose_trans(ref_frame,p[0.017635, 0.059017, 0.005000, -0.000000, 3.141593, -0.000000]),accel_mss,speed_ms,0,0) # end trace
    |   speed_ms    = 0.002
    |   movel(pose_trans(ref_frame,p[0.017635, 0.059017, -0.000125, -0.000000, 3.141593, -0.000000]),accel_mss,speed_ms,0,0) # end trace
    |   speed_ms    = 0.007
    |   movel(pose_trans(ref_frame,p[0.017700, 0.060806, -0.000125, -0.000000, 3.141593, -0.000000]),accel_mss,speed_ms,0,0.001)
    |   movel(pose_trans(ref_frame,p[0.018178, 0.062531, -0.000125, -0.000000, 3.141593, -0.000000]),accel_mss,speed_ms,0,0.001)
    |   movel(pose_trans(ref_frame,p[0.018153, 0.061894, -0.000125, -0.000000, 3.141593, -0.000000]),accel_mss,speed_ms,0,0.001)
    |   movel(pose_trans(ref_frame,p[0.018674, 0.061523, -0.000125, 0.000000, 3.141593, 0.000000]),accel_mss,speed_ms,0,0.001)
    |   movel(pose_trans(ref_frame,p[0.019204, 0.061987, -0.000125, -0.000000, 3.141593, 0.000000]),accel_mss,speed_ms,0,0.001)
    |   movel(pose_trans(ref_frame,p[0.019438, 0.062640, -0.000125, 0.000000, 3.141593, 0.000000]),accel_mss,speed_ms,0,0.001)
    |   movel(pose_trans(ref_frame,p[0.020702, 0.064436, -0.000125, -0.000000, 3.141593, -0.000000]),accel_mss,speed_ms,0,0.001)
    |   movel(pose_trans(ref_frame,p[0.021804, 0.066466, -0.000125, -0.000000, 3.141593, -0.000000]),accel_mss,speed_ms,0,0.001)
    |   movel(pose_trans(ref_frame,p[0.021509, 0.064697, -0.000125, 0.000000, 3.141593, -0.000000]),accel_mss,speed_ms,0,0.001)
    |   movel(pose_trans(ref_frame,p[0.021400, 0.063151, -0.000125, -0.000000, 3.141593, -0.000000]),accel_mss,speed_ms,0,0.001)
    |   movel(pose_trans(ref_frame,p[0.021961, 0.064210, -0.000125, 0.000000, 3.141593, 0.000000]),accel_mss,speed_ms,0,0.001)
    |   movel(pose_trans(ref_frame,p[0.022785, 0.065090, -0.000125, -0.000000, 3.141593, -0.000000]),accel_mss,speed_ms,0,0.001)
    |   movel(pose_trans(ref_frame,p[0.022476, 0.064068, -0.000125, 0.000000, 3.141593, -0.000000]),accel_mss,speed_ms,0,0.001)
    |   movel(pose_trans(ref_frame,p[0.022495, 0.063001, -0.000125, 0.000000, 3.141593, -0.000000]),accel_mss,speed_ms,0,0.001)
    |   movel(pose_trans(ref_frame,p[0.023403, 0.063152, -0.000125, 0.000000, 3.141593, -0.000000]),accel_mss,speed_ms,0,0.001)
    |   movel(pose_trans(ref_frame,p[0.024322, 0.063102, -0.000125, 0.000000, 3.141593, -0.000000]),accel_mss,speed_ms,0,0.001)
    |   movel(pose_trans(ref_frame,p[0.023261, 0.062612, -0.000125, 0.000000, 3.141593, -0.000000]),accel_mss,speed_ms,0,0.001)
    |   movel(pose_trans(ref_frame,p[0.022453, 0.061732, -0.000125, 0.000000, 3.141593, -0.000000]),accel_mss,speed_ms,0,0.001)
    |   movel(pose_trans(ref_frame,p[0.021865, 0.060700, -0.000125, -0.000000, 3.141593, 0.000000]),accel_mss,speed_ms,0,0.001)
    |   movel(pose_trans(ref_frame,p[0.021333, 0.059634, -0.000125, 0.000000, 3.141593, 0.000000]),accel_mss,speed_ms,0,0.001)
    |   movel(pose_trans(ref_frame,p[0.020337, 0.057910, -0.000125, 0.000000, 3.141593, -0.000000]),accel_mss,speed_ms,0,0.001)
    |   movel(pose_trans(ref_frame,p[0.018808, 0.056621, -0.000125, 0.000000, 3.141593, -0.000000]),accel_mss,speed_ms,0,0.001)
    |   movel(pose_trans(ref_frame,p[0.018010, 0.056489, -0.000125, -0.000000, 3.141593, 0.000000]),accel_mss,speed_ms,0,0.001)
    |   movel(pose_trans(ref_frame,p[0.017252, 0.056686, -0.000125, 0.000000, 3.141593, 0.000000]),accel_mss,speed_ms,0,0.001)
    |   movel(pose_trans(ref_frame,p[0.017003, 0.056829, -0.000125, -0.000000, 3.141593, -0.000000]),accel_mss,speed_ms,0,0.001)
    |   movel(pose_trans(ref_frame,p[0.016833, 0.057044, -0.000125, 0.000000, 3.141593, 0.000000]),accel_mss,speed_ms,0,0.001)
    |   movel(pose_trans(ref_frame,p[0.016894, 0.057464, -0.000125, -0.000000, 3.141593, -0.000000]),accel_mss,speed_ms,0,0.001)
    |   movel(pose_trans(ref_frame,p[0.017227, 0.057811, -0.000125, 0.000000, 3.141593, -0.000000]),accel_mss,speed_ms,0,0.001)
    |   movel(pose_trans(ref_frame,p[0.018459, 0.058742, -0.000125, 0.000000, 3.141593, -0.000000]),accel_mss,speed_ms,0,0.001)
    |   movel(pose_trans(ref_frame,p[0.019598, 0.059764, -0.000125, -0.000000, 3.141593, 0.000000]),accel_mss,speed_ms,0,0.001)
    |   movel(pose_trans(ref_frame,p[0.020174, 0.060624, -0.000125, -0.000000, 3.141593, -0.000000]),accel_mss,speed_ms,0,0.001)
    |   movel(pose_trans(ref_frame,p[0.020848, 0.061459, -0.000125, -0.000000, 3.141593, -0.000000]),accel_mss,speed_ms,0,0) # end trace
    |   speed_ms    = 1.000
    |   movel(pose_trans(ref_frame,p[0.020848, 0.061459, 0.005000, -0.000000, 3.141593, 0.000000]),accel_mss,speed_ms,0,0.001)
    |   movel(pose_trans(ref_frame,p[0.016658, 0.059526, 0.005000, 0.000000, 3.141593, -0.000000]),accel_mss,speed_ms,0,0) # end trace
    |   speed_ms    = 0.002
    |   movel(pose_trans(ref_frame,p[0.016658, 0.059526, -0.000125, 0.000000, 3.141593, 0.000000]),accel_mss,speed_ms,0,0) # end trace
    |   speed_ms    = 0.007
    |   movel(pose_trans(ref_frame,p[0.016087, 0.059768, -0.000125, 0.000000, 3.141593, -0.000000]),accel_mss,speed_ms,0,0.001)
    |   movel(pose_trans(ref_frame,p[0.015708, 0.060206, -0.000125, -0.000000, 3.141593, 0.000000]),accel_mss,speed_ms,0,0.001)
    |   movel(pose_trans(ref_frame,p[0.015664, 0.060454, -0.000125, 0.000000, 3.141593, 0.000000]),accel_mss,speed_ms,0,0.001)
    |   movel(pose_trans(ref_frame,p[0.015667, 0.060710, -0.000125, -0.000000, 3.141593, 0.000000]),accel_mss,speed_ms,0,0.001)
    |   movel(pose_trans(ref_frame,p[0.015759, 0.062657, -0.000125, -0.000000, 3.141593, -0.000000]),accel_mss,speed_ms,0,0.001)
    |   movel(pose_trans(ref_frame,p[0.015851, 0.064603, -0.000125, 0.000000, 3.141593, 0.000000]),accel_mss,speed_ms,0,0.001)
    |   movel(pose_trans(ref_frame,p[0.015956, 0.065190, -0.000125, -0.000000, 3.141593, -0.000000]),accel_mss,speed_ms,0,0.001)
    |   movel(pose_trans(ref_frame,p[0.016343, 0.065529, -0.000125, 0.000000, 3.141593, 0.000000]),accel_mss,speed_ms,0,0.001)
    |   movel(pose_trans(ref_frame,p[0.016834, 0.065419, -0.000125, -0.000000, 3.141593, -0.000000]),accel_mss,speed_ms,0,0.001)
    |   movel(pose_trans(ref_frame,p[0.017323, 0.065326, -0.000125, 0.000000, 3.141593, 0.000000]),accel_mss,speed_ms,0,0.001)
    |   movel(pose_trans(ref_frame,p[0.017578, 0.065478, -0.000125, -0.000000, 3.141593, -0.000000]),accel_mss,speed_ms,0,0.001)
    |   movel(pose_trans(ref_frame,p[0.017786, 0.065709, -0.000125, 0.000000, 3.141593, -0.000000]),accel_mss,speed_ms,0,0.001)
    |   movel(pose_trans(ref_frame,p[0.019087, 0.066324, -0.000125, 0.000000, 3.141593, -0.000000]),accel_mss,speed_ms,0,0.001)
    |   movel(pose_trans(ref_frame,p[0.020440, 0.065835, -0.000125, 0.000000, 3.141593, -0.000000]),accel_mss,speed_ms,0,0) # end trace
    |   speed_ms    = 1.000
    |   movel(pose_trans(ref_frame,p[0.020440, 0.065835, 0.005000, 0.000000, 3.141593, 0.000000]),accel_mss,speed_ms,0,0.001)
    |   movel(pose_trans(ref_frame,p[0.015991, 0.067324, 0.005000, 0.000000, 3.141593, 0.000000]),accel_mss,speed_ms,0,0) # end trace
    |   speed_ms    = 0.002
    |   movel(pose_trans(ref_frame,p[0.015991, 0.067324, -0.000125, 0.000000, 3.141593, 0.000000]),accel_mss,speed_ms,0,0) # end trace
    |   speed_ms    = 0.007
    |   movel(pose_trans(ref_frame,p[0.014334, 0.070841, -0.000125, -0.000000, 3.141593, 0.000000]),accel_mss,speed_ms,0,0.001)
    |   movel(pose_trans(ref_frame,p[0.014172, 0.071289, -0.000125, 0.000000, 3.141593, -0.000000]),accel_mss,speed_ms,0,0.001)
    |   movel(pose_trans(ref_frame,p[0.014241, 0.071722, -0.000125, 0.000000, 3.141593, -0.000000]),accel_mss,speed_ms,0,0.001)
    |   movel(pose_trans(ref_frame,p[0.014406, 0.071904, -0.000125, 0.000000, 3.141593, -0.000000]),accel_mss,speed_ms,0,0.001)
    |   movel(pose_trans(ref_frame,p[0.014552, 0.072096, -0.000125, -0.000000, 3.141593, 0.000000]),accel_mss,speed_ms,0,0.001)
    |   movel(pose_trans(ref_frame,p[0.014578, 0.072337, -0.000125, -0.000000, 3.141593, 0.000000]),accel_mss,speed_ms,0,0.001)
    |   movel(pose_trans(ref_frame,p[0.014501, 0.072578, -0.000125, 0.000000, 3.141593, 0.000000]),accel_mss,speed_ms,0,0.001)
    |   movel(pose_trans(ref_frame,p[0.013935, 0.073248, -0.000125, -0.000000, 3.141593, -0.000000]),accel_mss,speed_ms,0,0.001)
    |   movel(pose_trans(ref_frame,p[0.013240, 0.073777, -0.000125, -0.000000, 3.141593, -0.000000]),accel_mss,speed_ms,0,0.001)
    |   movel(pose_trans(ref_frame,p[0.012178, 0.074637, -0.000125, 0.000000, 3.141593, -0.000000]),accel_mss,speed_ms,0,0.001)
    |   movel(pose_trans(ref_frame,p[0.012560, 0.075688, -0.000125, -0.000000, 3.141593, 0.000000]),accel_mss,speed_ms,0,0.001)
    |   movel(pose_trans(ref_frame,p[0.011805, 0.076954, -0.000125, -0.000000, 3.141593, -0.000000]),accel_mss,speed_ms,0,0.001)
    |   movel(pose_trans(ref_frame,p[0.010607, 0.077857, -0.000125, 0.000000, 3.141593, -0.000000]),accel_mss,speed_ms,0,0.001)
    |   movel(pose_trans(ref_frame,p[0.009277, 0.078603, -0.000125, 0.000000, 3.141593, -0.000000]),accel_mss,speed_ms,0,0.001)
    |   movel(pose_trans(ref_frame,p[0.008159, 0.079596, -0.000125, 0.000000, 3.141593, 0.000000]),accel_mss,speed_ms,0,0.001)
    |   movel(pose_trans(ref_frame,p[0.008074, 0.079968, -0.000125, -0.000000, 3.141593, 0.000000]),accel_mss,speed_ms,0,0.001)
    |   movel(pose_trans(ref_frame,p[0.008272, 0.080211, -0.000125, -0.000000, 3.141593, -0.000000]),accel_mss,speed_ms,0,0.001)
    |   movel(pose_trans(ref_frame,p[0.008410, 0.080207, -0.000125, -0.000000, 3.141593, -0.000000]),accel_mss,speed_ms,0,0.001)
    |   movel(pose_trans(ref_frame,p[0.008543, 0.080159, -0.000125, 0.000000, 3.141593, 0.000000]),accel_mss,speed_ms,0,0.001)
    |   movel(pose_trans(ref_frame,p[0.009743, 0.079556, -0.000125, 0.000000, 3.141593, -0.000000]),accel_mss,speed_ms,0,0.001)
    |   movel(pose_trans(ref_frame,p[0.010863, 0.078815, -0.000125, -0.000000, 3.141593, -0.000000]),accel_mss,speed_ms,0,0.001)
    |   movel(pose_trans(ref_frame,p[0.010230, 0.080518, -0.000125, 0.000000, 3.141593, -0.000000]),accel_mss,speed_ms,0,0.001)
    |   movel(pose_trans(ref_frame,p[0.008545, 0.081520, -0.000125, -0.000000, 3.141593, 0.000000]),accel_mss,speed_ms,0,0.001)
    |   movel(pose_trans(ref_frame,p[0.008298, 0.081721, -0.000125, 0.000000, 3.141593, -0.000000]),accel_mss,speed_ms,0,0.001)
    |   movel(pose_trans(ref_frame,p[0.008194, 0.081991, -0.000125, -0.000000, 3.141593, -0.000000]),accel_mss,speed_ms,0,0.001)
    |   movel(pose_trans(ref_frame,p[0.008659, 0.082258, -0.000125, -0.000000, 3.141593, -0.000000]),accel_mss,speed_ms,0,0.001)
    |   movel(pose_trans(ref_frame,p[0.008980, 0.082386, -0.000125, 0.000000, 3.141593, -0.000000]),accel_mss,speed_ms,0,0.001)
    |   movel(pose_trans(ref_frame,p[0.008774, 0.083013, -0.000125, 0.000000, 3.141593, 0.000000]),accel_mss,speed_ms,0,0.001)
    |   movel(pose_trans(ref_frame,p[0.008213, 0.083462, -0.000125, -0.000000, 3.141593, 0.000000]),accel_mss,speed_ms,0,0.001)
    |   movel(pose_trans(ref_frame,p[0.007064, 0.084443, -0.000125, 0.000000, 3.141593, 0.000000]),accel_mss,speed_ms,0,0.001)
    |   movel(pose_trans(ref_frame,p[0.005896, 0.085402, -0.000125, -0.000000, 3.141593, -0.000000]),accel_mss,speed_ms,0,0.001)
    |   movel(pose_trans(ref_frame,p[0.005512, 0.085878, -0.000125, 0.000000, 3.141593, -0.000000]),accel_mss,speed_ms,0,0.001)
    |   movel(pose_trans(ref_frame,p[0.005552, 0.086389, -0.000125, 0.000000, 3.141593, 0.000000]),accel_mss,speed_ms,0,0.001)
    |   movel(pose_trans(ref_frame,p[0.006014, 0.086548, -0.000125, -0.000000, 3.141593, 0.000000]),accel_mss,speed_ms,0,0.001)
    |   movel(pose_trans(ref_frame,p[0.006546, 0.086337, -0.000125, 0.000000, 3.141593, 0.000000]),accel_mss,speed_ms,0,0.001)
    |   movel(pose_trans(ref_frame,p[0.009369, 0.084529, -0.000125, -0.000000, 3.141593, -0.000000]),accel_mss,speed_ms,0,0.001)
    |   movel(pose_trans(ref_frame,p[0.012003, 0.082456, -0.000125, -0.000000, 3.141593, 0.000000]),accel_mss,speed_ms,0,0.001)
    |   movel(pose_trans(ref_frame,p[0.012459, 0.082035, -0.000125, 0.000000, 3.141593, -0.000000]),accel_mss,speed_ms,0,0.001)
    |   movel(pose_trans(ref_frame,p[0.012849, 0.081558, -0.000125, -0.000000, 3.141593, -0.000000]),accel_mss,speed_ms,0,0.001)
    |   movel(pose_trans(ref_frame,p[0.013160, 0.080901, -0.000125, 0.000000, 3.141593, -0.000000]),accel_mss,speed_ms,0,0.001)
    |   movel(pose_trans(ref_frame,p[0.013366, 0.080198, -0.000125, -0.000000, 3.141593, -0.000000]),accel_mss,speed_ms,0,0.001)
    |   movel(pose_trans(ref_frame,p[0.013644, 0.077586, -0.000125, -0.000000, 3.141593, 0.000000]),accel_mss,speed_ms,0,0.001)
    |   movel(pose_trans(ref_frame,p[0.015097, 0.075575, -0.000125, 0.000000, 3.141593, 0.000000]),accel_mss,speed_ms,0,0.001)
    |   movel(pose_trans(ref_frame,p[0.015507, 0.075506, -0.000125, 0.000000, 3.141593, 0.000000]),accel_mss,speed_ms,0,0.001)
    |   movel(pose_trans(ref_frame,p[0.015858, 0.075341, -0.000125, 0.000000, 3.141593, 0.000000]),accel_mss,speed_ms,0,0.001)
    |   movel(pose_trans(ref_frame,p[0.015980, 0.075081, -0.000125, -0.000000, 3.141593, -0.000000]),accel_mss,speed_ms,0,0.001)
    |   movel(pose_trans(ref_frame,p[0.015998, 0.074782, -0.000125, -0.000000, 3.141593, 0.000000]),accel_mss,speed_ms,0,0.001)
    |   movel(pose_trans(ref_frame,p[0.016404, 0.071019, -0.000125, -0.000000, 3.141593, 0.000000]),accel_mss,speed_ms,0,0.001)
    |   movel(pose_trans(ref_frame,p[0.017386, 0.067303, -0.000125, -0.000000, 3.141593, 0.000000]),accel_mss,speed_ms,0,0) # end trace
    |   speed_ms    = 1.000
    |   movel(pose_trans(ref_frame,p[0.017386, 0.067303, 0.005000, -0.000000, 3.141593, 0.000000]),accel_mss,speed_ms,0,0.001)
    |   movel(pose_trans(ref_frame,p[0.017926, 0.070135, 0.005000, -0.000000, 3.141593, -0.000000]),accel_mss,speed_ms,0,0) # end trace
    |   speed_ms    = 0.002
    |   movel(pose_trans(ref_frame,p[0.017926, 0.070135, -0.000125, -0.000000, 3.141593, 0.000000]),accel_mss,speed_ms,0,0) # end trace
    |   speed_ms    = 0.007
    |   movel(pose_trans(ref_frame,p[0.018156, 0.072084, -0.000125, 0.000000, 3.141593, 0.000000]),accel_mss,speed_ms,0,0.001)
    |   movel(pose_trans(ref_frame,p[0.018548, 0.074007, -0.000125, 0.000000, 3.141593, -0.000000]),accel_mss,speed_ms,0,0.001)
    |   movel(pose_trans(ref_frame,p[0.018828, 0.073764, -0.000125, 0.000000, 3.141593, -0.000000]),accel_mss,speed_ms,0,0.001)
    |   movel(pose_trans(ref_frame,p[0.019109, 0.073521, -0.000125, -0.000000, 3.141593, 0.000000]),accel_mss,speed_ms,0,0.001)
    |   movel(pose_trans(ref_frame,p[0.019211, 0.073447, -0.000125, -0.000000, 3.141593, 0.000000]),accel_mss,speed_ms,0,0.001)
    |   movel(pose_trans(ref_frame,p[0.019327, 0.073430, -0.000125, 0.000000, 3.141593, -0.000000]),accel_mss,speed_ms,0,0.001)
    |   movel(pose_trans(ref_frame,p[0.019423, 0.073501, -0.000125, 0.000000, 3.141593, -0.000000]),accel_mss,speed_ms,0,0.001)
    |   movel(pose_trans(ref_frame,p[0.019480, 0.073617, -0.000125, 0.000000, 3.141593, 0.000000]),accel_mss,speed_ms,0,0.001)
    |   movel(pose_trans(ref_frame,p[0.019837, 0.074328, -0.000125, -0.000000, 3.141593, 0.000000]),accel_mss,speed_ms,0,0.001)
    |   movel(pose_trans(ref_frame,p[0.020311, 0.074967, -0.000125, -0.000000, 3.141593, -0.000000]),accel_mss,speed_ms,0,0.001)
    |   movel(pose_trans(ref_frame,p[0.020450, 0.075091, -0.000125, 0.000000, 3.141593, 0.000000]),accel_mss,speed_ms,0,0.001)
    |   movel(pose_trans(ref_frame,p[0.020616, 0.075117, -0.000125, 0.000000, 3.141593, -0.000000]),accel_mss,speed_ms,0,0.001)
    |   movel(pose_trans(ref_frame,p[0.020728, 0.075021, -0.000125, 0.000000, 3.141593, -0.000000]),accel_mss,speed_ms,0,0.001)
    |   movel(pose_trans(ref_frame,p[0.020786, 0.074874, -0.000125, -0.000000, 3.141593, -0.000000]),accel_mss,speed_ms,0,0.001)
    |   movel(pose_trans(ref_frame,p[0.020978, 0.073939, -0.000125, -0.000000, 3.141593, -0.000000]),accel_mss,speed_ms,0,0.001)
    |   movel(pose_trans(ref_frame,p[0.021025, 0.072985, -0.000125, -0.000000, 3.141593, -0.000000]),accel_mss,speed_ms,0,0) # end trace
    |   speed_ms    = 1.000
    |   movel(pose_trans(ref_frame,p[0.021025, 0.072985, 0.005000, -0.000000, 3.141593, 0.000000]),accel_mss,speed_ms,0,0.001)
    |   movel(pose_trans(ref_frame,p[0.019272, 0.075044, 0.005000, 0.000000, 3.141593, 0.000000]),accel_mss,speed_ms,0,0) # end trace
    |   speed_ms    = 0.002
    |   movel(pose_trans(ref_frame,p[0.019272, 0.075044, -0.000125, 0.000000, 3.141593, -0.000000]),accel_mss,speed_ms,0,0) # end trace
    |   speed_ms    = 0.007
    |   movel(pose_trans(ref_frame,p[0.019280, 0.077860, -0.000125, -0.000000, 3.141593, -0.000000]),accel_mss,speed_ms,0,0.001)
    |   movel(pose_trans(ref_frame,p[0.020023, 0.080577, -0.000125, 0.000000, 3.141593, 0.000000]),accel_mss,speed_ms,0,0.001)
    |   movel(pose_trans(ref_frame,p[0.020120, 0.079640, -0.000125, 0.000000, 3.141593, 0.000000]),accel_mss,speed_ms,0,0.001)
    |   movel(pose_trans(ref_frame,p[0.020687, 0.078888, -0.000125, -0.000000, 3.141593, -0.000000]),accel_mss,speed_ms,0,0) # end trace
    |   speed_ms    = 1.000
    |   movel(pose_trans(ref_frame,p[0.020687, 0.078888, 0.005000, -0.000000, 3.141593, 0.000000]),accel_mss,speed_ms,0,0.001)
    |   movel(pose_trans(ref_frame,p[0.013058, 0.060216, 0.005000, -0.000000, 3.141593, -0.000000]),accel_mss,speed_ms,0,0) # end trace
    |   speed_ms    = 0.002
    |   movel(pose_trans(ref_frame,p[0.013058, 0.060216, -0.000125, -0.000000, 3.141593, -0.000000]),accel_mss,speed_ms,0,0) # end trace
    |   speed_ms    = 0.007
    |   movel(pose_trans(ref_frame,p[0.012127, 0.060528, -0.000125, 0.000000, 3.141593, -0.000000]),accel_mss,speed_ms,0,0.001)
    |   movel(pose_trans(ref_frame,p[0.011433, 0.061217, -0.000125, 0.000000, 3.141593, -0.000000]),accel_mss,speed_ms,0,0.001)
    |   movel(pose_trans(ref_frame,p[0.011357, 0.060164, -0.000125, -0.000000, 3.141593, 0.000000]),accel_mss,speed_ms,0,0.001)
    |   movel(pose_trans(ref_frame,p[0.011321, 0.059025, -0.000125, -0.000000, 3.141593, -0.000000]),accel_mss,speed_ms,0,0.001)
    |   movel(pose_trans(ref_frame,p[0.011572, 0.057982, -0.000125, -0.000000, 3.141593, -0.000000]),accel_mss,speed_ms,0,0.001)
    |   movel(pose_trans(ref_frame,p[0.012191, 0.057184, -0.000125, -0.000000, 3.141593, -0.000000]),accel_mss,speed_ms,0,0.001)
    |   movel(pose_trans(ref_frame,p[0.011997, 0.057795, -0.000125, 0.000000, 3.141593, -0.000000]),accel_mss,speed_ms,0,0.001)
    |   movel(pose_trans(ref_frame,p[0.012167, 0.058415, -0.000125, -0.000000, 3.141593, 0.000000]),accel_mss,speed_ms,0,0.001)
    |   movel(pose_trans(ref_frame,p[0.012454, 0.057908, -0.000125, 0.000000, 3.141593, -0.000000]),accel_mss,speed_ms,0,0.001)
    |   movel(pose_trans(ref_frame,p[0.012859, 0.057512, -0.000125, -0.000000, 3.141593, 0.000000]),accel_mss,speed_ms,0,0.001)
    |   movel(pose_trans(ref_frame,p[0.013428, 0.057397, -0.000125, 0.000000, 3.141593, -0.000000]),accel_mss,speed_ms,0,0.001)
    |   movel(pose_trans(ref_frame,p[0.013858, 0.057722, -0.000125, -0.000000, 3.141593, -0.000000]),accel_mss,speed_ms,0,0) # end trace
    |   speed_ms    = 1.000
    |   movel(pose_trans(ref_frame,p[0.013858, 0.057722, 0.005000, -0.000000, 3.141593, -0.000000]),accel_mss,speed_ms,0,0.001)
    |   movel(pose_trans(ref_frame,p[0.015336, 0.056324, 0.005000, -0.000000, 3.141593, -0.000000]),accel_mss,speed_ms,0,0) # end trace
    |   speed_ms    = 0.002
    |   movel(pose_trans(ref_frame,p[0.015336, 0.056324, -0.000125, -0.000000, 3.141593, 0.000000]),accel_mss,speed_ms,0,0) # end trace
    |   speed_ms    = 0.007
    |   movel(pose_trans(ref_frame,p[0.015028, 0.056519, -0.000125, -0.000000, 3.141593, 0.000000]),accel_mss,speed_ms,0,0.001)
    |   movel(pose_trans(ref_frame,p[0.014778, 0.056775, -0.000125, -0.000000, 3.141593, 0.000000]),accel_mss,speed_ms,0,0.001)
    |   movel(pose_trans(ref_frame,p[0.014670, 0.057124, -0.000125, 0.000000, 3.141593, -0.000000]),accel_mss,speed_ms,0,0.001)
    |   movel(pose_trans(ref_frame,p[0.014805, 0.057442, -0.000125, 0.000000, 3.141593, -0.000000]),accel_mss,speed_ms,0,0.001)
    |   movel(pose_trans(ref_frame,p[0.014939, 0.057536, -0.000125, -0.000000, 3.141593, -0.000000]),accel_mss,speed_ms,0,0.001)
    |   movel(pose_trans(ref_frame,p[0.015066, 0.057636, -0.000125, 0.000000, 3.141593, -0.000000]),accel_mss,speed_ms,0,0.001)
    |   movel(pose_trans(ref_frame,p[0.015154, 0.057950, -0.000125, 0.000000, 3.141593, -0.000000]),accel_mss,speed_ms,0,0.001)
    |   movel(pose_trans(ref_frame,p[0.015037, 0.058289, -0.000125, -0.000000, 3.141593, 0.000000]),accel_mss,speed_ms,0,0.001)
    |   movel(pose_trans(ref_frame,p[0.014542, 0.058958, -0.000125, 0.000000, 3.141593, -0.000000]),accel_mss,speed_ms,0,0.001)
    |   movel(pose_trans(ref_frame,p[0.013874, 0.059455, -0.000125, -0.000000, 3.141593, 0.000000]),accel_mss,speed_ms,0,0.001)
    |   movel(pose_trans(ref_frame,p[0.014214, 0.060874, -0.000125, -0.000000, 3.141593, 0.000000]),accel_mss,speed_ms,0,0.001)
    |   movel(pose_trans(ref_frame,p[0.013874, 0.062379, -0.000125, 0.000000, 3.141593, 0.000000]),accel_mss,speed_ms,0,0.001)
    |   movel(pose_trans(ref_frame,p[0.013650, 0.063093, -0.000125, -0.000000, 3.141593, 0.000000]),accel_mss,speed_ms,0,0.001)
    |   movel(pose_trans(ref_frame,p[0.013602, 0.063824, -0.000125, -0.000000, 3.141593, 0.000000]),accel_mss,speed_ms,0,0.001)
    |   movel(pose_trans(ref_frame,p[0.013933, 0.064493, -0.000125, -0.000000, 3.141593, 0.000000]),accel_mss,speed_ms,0,0.001)
    |   movel(pose_trans(ref_frame,p[0.014596, 0.064710, -0.000125, -0.000000, 3.141593, -0.000000]),accel_mss,speed_ms,0,0.001)
    |   movel(pose_trans(ref_frame,p[0.014021, 0.066041, -0.000125, 0.000000, 3.141593, -0.000000]),accel_mss,speed_ms,0,0.001)
    |   movel(pose_trans(ref_frame,p[0.014179, 0.067482, -0.000125, -0.000000, 3.141593, -0.000000]),accel_mss,speed_ms,0,0) # end trace
    |   speed_ms    = 1.000
    |   movel(pose_trans(ref_frame,p[0.014179, 0.067482, 0.005000, -0.000000, 3.141593, -0.000000]),accel_mss,speed_ms,0,0.001)
    |   movel(pose_trans(ref_frame,p[0.002339, 0.066901, 0.005000, -0.000000, 3.141593, -0.000000]),accel_mss,speed_ms,0,0) # end trace
    |   speed_ms    = 0.002
    |   movel(pose_trans(ref_frame,p[0.002339, 0.066901, -0.000125, -0.000000, 3.141593, -0.000000]),accel_mss,speed_ms,0,0) # end trace
    |   speed_ms    = 0.007
    |   movel(pose_trans(ref_frame,p[0.003951, 0.065057, -0.000125, 0.000000, 3.141593, -0.000000]),accel_mss,speed_ms,0,0.001)
    |   movel(pose_trans(ref_frame,p[0.006316, 0.064421, -0.000125, 0.000000, 3.141593, -0.000000]),accel_mss,speed_ms,0,0.001)
    |   movel(pose_trans(ref_frame,p[0.008466, 0.064760, -0.000125, -0.000000, 3.141593, -0.000000]),accel_mss,speed_ms,0,0.001)
    |   movel(pose_trans(ref_frame,p[0.010502, 0.064577, -0.000125, -0.000000, 3.141593, -0.000000]),accel_mss,speed_ms,0,0.001)
    |   movel(pose_trans(ref_frame,p[0.011572, 0.063544, -0.000125, -0.000000, 3.141593, -0.000000]),accel_mss,speed_ms,0,0.001)
    |   movel(pose_trans(ref_frame,p[0.012146, 0.062104, -0.000125, -0.000000, 3.141593, -0.000000]),accel_mss,speed_ms,0,0) # end trace
    |   speed_ms    = 1.000
    |   movel(pose_trans(ref_frame,p[0.012146, 0.062104, 0.005000, -0.000000, 3.141593, 0.000000]),accel_mss,speed_ms,0,0.001)
    |   movel(pose_trans(ref_frame,p[0.012580, 0.048770, 0.005000, -0.000000, 3.141593, -0.000000]),accel_mss,speed_ms,0,0) # end trace
    |   speed_ms    = 0.002
    |   movel(pose_trans(ref_frame,p[0.012580, 0.048770, -0.000125, -0.000000, 3.141593, 0.000000]),accel_mss,speed_ms,0,0) # end trace
    |   speed_ms    = 0.007
    |   movel(pose_trans(ref_frame,p[0.012449, 0.049200, -0.000125, 0.000000, 3.141593, -0.000000]),accel_mss,speed_ms,0,0.001)
    |   movel(pose_trans(ref_frame,p[0.012655, 0.049627, -0.000125, 0.000000, 3.141593, 0.000000]),accel_mss,speed_ms,0,0.001)
    |   movel(pose_trans(ref_frame,p[0.013153, 0.049876, -0.000125, -0.000000, 3.141593, -0.000000]),accel_mss,speed_ms,0,0.001)
    |   movel(pose_trans(ref_frame,p[0.013599, 0.050072, -0.000125, -0.000000, 3.141593, -0.000000]),accel_mss,speed_ms,0,0.001)
    |   movel(pose_trans(ref_frame,p[0.013770, 0.050361, -0.000125, 0.000000, 3.141593, -0.000000]),accel_mss,speed_ms,0,0.001)
    |   movel(pose_trans(ref_frame,p[0.013962, 0.050694, -0.000125, -0.000000, 3.141593, -0.000000]),accel_mss,speed_ms,0,0.001)
    |   movel(pose_trans(ref_frame,p[0.014849, 0.051248, -0.000125, 0.000000, 3.141593, 0.000000]),accel_mss,speed_ms,0,0.001)
    |   movel(pose_trans(ref_frame,p[0.015857, 0.051500, -0.000125, -0.000000, 3.141593, 0.000000]),accel_mss,speed_ms,0,0.001)
    |   movel(pose_trans(ref_frame,p[0.015592, 0.051422, -0.000125, 0.000000, 3.141593, 0.000000]),accel_mss,speed_ms,0,0.001)
    |   movel(pose_trans(ref_frame,p[0.015321, 0.051389, -0.000125, 0.000000, 3.141593, 0.000000]),accel_mss,speed_ms,0,0.001)
    |   movel(pose_trans(ref_frame,p[0.015051, 0.051446, -0.000125, -0.000000, 3.141593, 0.000000]),accel_mss,speed_ms,0,0.001)
    |   movel(pose_trans(ref_frame,p[0.014846, 0.051621, -0.000125, 0.000000, 3.141593, -0.000000]),accel_mss,speed_ms,0,0.001)
    |   movel(pose_trans(ref_frame,p[0.014775, 0.051875, -0.000125, 0.000000, 3.141593, 0.000000]),accel_mss,speed_ms,0,0.001)
    |   movel(pose_trans(ref_frame,p[0.014834, 0.052136, -0.000125, -0.000000, 3.141593, -0.000000]),accel_mss,speed_ms,0,0.001)
    |   movel(pose_trans(ref_frame,p[0.014984, 0.052357, -0.000125, -0.000000, 3.141593, -0.000000]),accel_mss,speed_ms,0,0.001)
    |   movel(pose_trans(ref_frame,p[0.015182, 0.052541, -0.000125, -0.000000, 3.141593, 0.000000]),accel_mss,speed_ms,0,0.001)
    |   movel(pose_trans(ref_frame,p[0.015912, 0.052995, -0.000125, 0.000000, 3.141593, 0.000000]),accel_mss,speed_ms,0,0.001)
    |   movel(pose_trans(ref_frame,p[0.016735, 0.053246, -0.000125, 0.000000, 3.141593, 0.000000]),accel_mss,speed_ms,0,0.001)
    |   movel(pose_trans(ref_frame,p[0.015727, 0.053094, -0.000125, 0.000000, 3.141593, -0.000000]),accel_mss,speed_ms,0,0.001)
    |   movel(pose_trans(ref_frame,p[0.014783, 0.053002, -0.000125, -0.000000, 3.141593, -0.000000]),accel_mss,speed_ms,0,0.001)
    |   movel(pose_trans(ref_frame,p[0.014704, 0.053020, -0.000125, -0.000000, 3.141593, 0.000000]),accel_mss,speed_ms,0,0.001)
    |   movel(pose_trans(ref_frame,p[0.014639, 0.053062, -0.000125, 0.000000, 3.141593, 0.000000]),accel_mss,speed_ms,0,0.001)
    |   movel(pose_trans(ref_frame,p[0.014610, 0.053165, -0.000125, -0.000000, 3.141593, 0.000000]),accel_mss,speed_ms,0,0.001)
    |   movel(pose_trans(ref_frame,p[0.014639, 0.053278, -0.000125, -0.000000, 3.141593, -0.000000]),accel_mss,speed_ms,0,0.001)
    |   movel(pose_trans(ref_frame,p[0.014964, 0.053829, -0.000125, -0.000000, 3.141593, -0.000000]),accel_mss,speed_ms,0,0.001)
    |   movel(pose_trans(ref_frame,p[0.015445, 0.054249, -0.000125, 0.000000, 3.141593, -0.000000]),accel_mss,speed_ms,0,0.001)
    |   movel(pose_trans(ref_frame,p[0.013568, 0.054303, -0.000125, 0.000000, 3.141593, -0.000000]),accel_mss,speed_ms,0,0.001)
    |   movel(pose_trans(ref_frame,p[0.013884, 0.055693, -0.000125, 0.000000, 3.141593, -0.000000]),accel_mss,speed_ms,0,0.001)
    |   movel(pose_trans(ref_frame,p[0.014121, 0.055690, -0.000125, 0.000000, 3.141593, -0.000000]),accel_mss,speed_ms,0,0.001)
    |   movel(pose_trans(ref_frame,p[0.014354, 0.055627, -0.000125, 0.000000, 3.141593, -0.000000]),accel_mss,speed_ms,0,0.001)
    |   movel(pose_trans(ref_frame,p[0.015085, 0.055350, -0.000125, 0.000000, 3.141593, 0.000000]),accel_mss,speed_ms,0,0.001)
    |   movel(pose_trans(ref_frame,p[0.015836, 0.055192, -0.000125, 0.000000, 3.141593, 0.000000]),accel_mss,speed_ms,0,0.001)
    |   movel(pose_trans(ref_frame,p[0.016463, 0.055275, -0.000125, 0.000000, 3.141593, -0.000000]),accel_mss,speed_ms,0,0.001)
    |   movel(pose_trans(ref_frame,p[0.017087, 0.055404, -0.000125, 0.000000, 3.141593, -0.000000]),accel_mss,speed_ms,0,0.001)
    |   movel(pose_trans(ref_frame,p[0.017732, 0.055357, -0.000125, 0.000000, 3.141593, 0.000000]),accel_mss,speed_ms,0,0.001)
    |   movel(pose_trans(ref_frame,p[0.018201, 0.054977, -0.000125, -0.000000, 3.141593, -0.000000]),accel_mss,speed_ms,0,0.001)
    |   movel(pose_trans(ref_frame,p[0.017947, 0.054692, -0.000125, -0.000000, 3.141593, -0.000000]),accel_mss,speed_ms,0,0.001)
    |   movel(pose_trans(ref_frame,p[0.017655, 0.054445, -0.000125, -0.000000, 3.141593, 0.000000]),accel_mss,speed_ms,0,0) # end trace
    |   speed_ms    = 1.000
    |   movel(pose_trans(ref_frame,p[0.017655, 0.054445, 0.005000, -0.000000, 3.141593, 0.000000]),accel_mss,speed_ms,0,0.001)
    |   movel(pose_trans(ref_frame,p[0.017079, 0.049540, 0.005000, -0.000000, 3.141593, 0.000000]),accel_mss,speed_ms,0,0) # end trace
    |   speed_ms    = 0.002
    |   movel(pose_trans(ref_frame,p[0.017079, 0.049540, -0.000125, -0.000000, 3.141593, 0.000000]),accel_mss,speed_ms,0,0) # end trace
    |   speed_ms    = 0.007
    |   movel(pose_trans(ref_frame,p[0.017725, 0.050203, -0.000125, -0.000000, 3.141593, -0.000000]),accel_mss,speed_ms,0,0.001)
    |   movel(pose_trans(ref_frame,p[0.018678, 0.050411, -0.000125, -0.000000, 3.141593, 0.000000]),accel_mss,speed_ms,0,0.001)
    |   movel(pose_trans(ref_frame,p[0.019636, 0.050317, -0.000125, -0.000000, 3.141593, 0.000000]),accel_mss,speed_ms,0,0.001)
    |   movel(pose_trans(ref_frame,p[0.020593, 0.050190, -0.000125, 0.000000, 3.141593, -0.000000]),accel_mss,speed_ms,0,0.001)
    |   movel(pose_trans(ref_frame,p[0.023132, 0.050771, -0.000125, -0.000000, 3.141593, 0.000000]),accel_mss,speed_ms,0,0.001)
    |   movel(pose_trans(ref_frame,p[0.025378, 0.052272, -0.000125, 0.000000, 3.141593, 0.000000]),accel_mss,speed_ms,0,0.001)
    |   movel(pose_trans(ref_frame,p[0.027522, 0.053904, -0.000125, -0.000000, 3.141593, 0.000000]),accel_mss,speed_ms,0,0.001)
    |   movel(pose_trans(ref_frame,p[0.029937, 0.054942, -0.000125, 0.000000, 3.141593, -0.000000]),accel_mss,speed_ms,0,0.001)
    |   movel(pose_trans(ref_frame,p[0.034741, 0.051742, -0.000125, -0.000000, 3.141593, -0.000000]),accel_mss,speed_ms,0,0.001)
    |   movel(pose_trans(ref_frame,p[0.034719, 0.046256, -0.000125, 0.000000, 3.141593, -0.000000]),accel_mss,speed_ms,0,0.001)
    |   movel(pose_trans(ref_frame,p[0.034180, 0.044195, -0.000125, -0.000000, 3.141593, 0.000000]),accel_mss,speed_ms,0,0.001)
    |   movel(pose_trans(ref_frame,p[0.033633, 0.042137, -0.000125, 0.000000, 3.141593, -0.000000]),accel_mss,speed_ms,0,0.001)
    |   movel(pose_trans(ref_frame,p[0.033137, 0.040165, -0.000125, -0.000000, 3.141593, 0.000000]),accel_mss,speed_ms,0,0.001)
    |   movel(pose_trans(ref_frame,p[0.033439, 0.038187, -0.000125, 0.000000, 3.141593, 0.000000]),accel_mss,speed_ms,0,0.001)
    |   movel(pose_trans(ref_frame,p[0.033960, 0.037638, -0.000125, 0.000000, 3.141593, 0.000000]),accel_mss,speed_ms,0,0.001)
    |   movel(pose_trans(ref_frame,p[0.034531, 0.037126, -0.000125, -0.000000, 3.141593, -0.000000]),accel_mss,speed_ms,0,0.001)
    |   movel(pose_trans(ref_frame,p[0.035000, 0.036281, -0.000125, -0.000000, 3.141593, 0.000000]),accel_mss,speed_ms,0,0.001)
    |   movel(pose_trans(ref_frame,p[0.035134, 0.035310, -0.000125, -0.000000, 3.141593, -0.000000]),accel_mss,speed_ms,0,0.001)
    |   movel(pose_trans(ref_frame,p[0.035022, 0.034342, -0.000125, 0.000000, 3.141593, -0.000000]),accel_mss,speed_ms,0,0.001)
    |   movel(pose_trans(ref_frame,p[0.034768, 0.033395, -0.000125, -0.000000, 3.141593, 0.000000]),accel_mss,speed_ms,0,0.001)
    |   movel(pose_trans(ref_frame,p[0.034179, 0.031720, -0.000125, -0.000000, 3.141593, -0.000000]),accel_mss,speed_ms,0,0.001)
    |   movel(pose_trans(ref_frame,p[0.033320, 0.030180, -0.000125, -0.000000, 3.141593, 0.000000]),accel_mss,speed_ms,0,0) # end trace
    |   speed_ms    = 1.000
    |   movel(pose_trans(ref_frame,p[0.033320, 0.030180, 0.005000, -0.000000, 3.141593, -0.000000]),accel_mss,speed_ms,0,0.001)
    |   movel(pose_trans(ref_frame,p[0.018489, 0.042386, 0.005000, -0.000000, 3.141593, -0.000000]),accel_mss,speed_ms,0,0) # end trace
    |   speed_ms    = 0.002
    |   movel(pose_trans(ref_frame,p[0.018489, 0.042386, -0.000125, -0.000000, 3.141593, -0.000000]),accel_mss,speed_ms,0,0) # end trace
    |   speed_ms    = 0.007
    |   movel(pose_trans(ref_frame,p[0.019483, 0.041896, -0.000125, 0.000000, 3.141593, -0.000000]),accel_mss,speed_ms,0,0.001)
    |   movel(pose_trans(ref_frame,p[0.020706, 0.041805, -0.000125, 0.000000, 3.141593, 0.000000]),accel_mss,speed_ms,0,0.001)
    |   movel(pose_trans(ref_frame,p[0.019991, 0.042414, -0.000125, 0.000000, 3.141593, -0.000000]),accel_mss,speed_ms,0,0.001)
    |   movel(pose_trans(ref_frame,p[0.019717, 0.043143, -0.000125, 0.000000, 3.141593, -0.000000]),accel_mss,speed_ms,0,0.001)
    |   movel(pose_trans(ref_frame,p[0.020836, 0.044174, -0.000125, 0.000000, 3.141593, -0.000000]),accel_mss,speed_ms,0,0.001)
    |   movel(pose_trans(ref_frame,p[0.021981, 0.045178, -0.000125, 0.000000, 3.141593, -0.000000]),accel_mss,speed_ms,0,0.001)
    |   movel(pose_trans(ref_frame,p[0.022455, 0.045361, -0.000125, -0.000000, 3.141593, 0.000000]),accel_mss,speed_ms,0,0.001)
    |   movel(pose_trans(ref_frame,p[0.023001, 0.045310, -0.000125, -0.000000, 3.141593, -0.000000]),accel_mss,speed_ms,0,0.001)
    |   movel(pose_trans(ref_frame,p[0.023530, 0.045215, -0.000125, 0.000000, 3.141593, -0.000000]),accel_mss,speed_ms,0,0.001)
    |   movel(pose_trans(ref_frame,p[0.024046, 0.045263, -0.000125, 0.000000, 3.141593, -0.000000]),accel_mss,speed_ms,0,0.001)
    |   movel(pose_trans(ref_frame,p[0.023757, 0.046397, -0.000125, -0.000000, 3.141593, -0.000000]),accel_mss,speed_ms,0,0.001)
    |   movel(pose_trans(ref_frame,p[0.023790, 0.047567, -0.000125, -0.000000, 3.141593, -0.000000]),accel_mss,speed_ms,0,0.001)
    |   movel(pose_trans(ref_frame,p[0.023945, 0.048228, -0.000125, -0.000000, 3.141593, -0.000000]),accel_mss,speed_ms,0,0.001)
    |   movel(pose_trans(ref_frame,p[0.024140, 0.048879, -0.000125, 0.000000, 3.141593, 0.000000]),accel_mss,speed_ms,0,0.001)
    |   movel(pose_trans(ref_frame,p[0.024355, 0.049667, -0.000125, 0.000000, 3.141593, -0.000000]),accel_mss,speed_ms,0,0.001)
    |   movel(pose_trans(ref_frame,p[0.024535, 0.050464, -0.000125, -0.000000, 3.141593, -0.000000]),accel_mss,speed_ms,0,0) # end trace
    |   speed_ms    = 1.000
    |   movel(pose_trans(ref_frame,p[0.024535, 0.050464, 0.005000, -0.000000, 3.141593, 0.000000]),accel_mss,speed_ms,0,0.001)
    |   movel(pose_trans(ref_frame,p[0.021815, 0.049337, 0.005000, 0.000000, 3.141593, 0.000000]),accel_mss,speed_ms,0,0) # end trace
    |   speed_ms    = 0.002
    |   movel(pose_trans(ref_frame,p[0.021815, 0.049337, -0.000125, 0.000000, 3.141593, 0.000000]),accel_mss,speed_ms,0,0) # end trace
    |   speed_ms    = 0.007
    |   movel(pose_trans(ref_frame,p[0.021581, 0.048363, -0.000125, -0.000000, 3.141593, -0.000000]),accel_mss,speed_ms,0,0.001)
    |   movel(pose_trans(ref_frame,p[0.021056, 0.047554, -0.000125, 0.000000, 3.141593, -0.000000]),accel_mss,speed_ms,0,0.001)
    |   movel(pose_trans(ref_frame,p[0.020463, 0.047211, -0.000125, -0.000000, 3.141593, 0.000000]),accel_mss,speed_ms,0,0.001)
    |   movel(pose_trans(ref_frame,p[0.019799, 0.046993, -0.000125, -0.000000, 3.141593, -0.000000]),accel_mss,speed_ms,0,0.001)
    |   movel(pose_trans(ref_frame,p[0.018812, 0.046368, -0.000125, 0.000000, 3.141593, -0.000000]),accel_mss,speed_ms,0,0.001)
    |   movel(pose_trans(ref_frame,p[0.018086, 0.045497, -0.000125, -0.000000, 3.141593, -0.000000]),accel_mss,speed_ms,0,0.001)
    |   movel(pose_trans(ref_frame,p[0.017267, 0.045028, -0.000125, 0.000000, 3.141593, 0.000000]),accel_mss,speed_ms,0,0.001)
    |   movel(pose_trans(ref_frame,p[0.016317, 0.044815, -0.000125, 0.000000, 3.141593, 0.000000]),accel_mss,speed_ms,0,0.001)
    |   movel(pose_trans(ref_frame,p[0.015348, 0.044468, -0.000125, -0.000000, 3.141593, -0.000000]),accel_mss,speed_ms,0,0.001)
    |   movel(pose_trans(ref_frame,p[0.014459, 0.043939, -0.000125, -0.000000, 3.141593, 0.000000]),accel_mss,speed_ms,0,0.001)
    |   movel(pose_trans(ref_frame,p[0.013987, 0.043237, -0.000125, -0.000000, 3.141593, -0.000000]),accel_mss,speed_ms,0,0.001)
    |   movel(pose_trans(ref_frame,p[0.014174, 0.042524, -0.000125, -0.000000, 3.141593, -0.000000]),accel_mss,speed_ms,0,0.001)
    |   movel(pose_trans(ref_frame,p[0.015942, 0.041840, -0.000125, -0.000000, 3.141593, -0.000000]),accel_mss,speed_ms,0,0.001)
    |   movel(pose_trans(ref_frame,p[0.017701, 0.042407, -0.000125, 0.000000, 3.141593, -0.000000]),accel_mss,speed_ms,0,0.001)
    |   movel(pose_trans(ref_frame,p[0.018133, 0.042814, -0.000125, -0.000000, 3.141593, -0.000000]),accel_mss,speed_ms,0,0.001)
    |   movel(pose_trans(ref_frame,p[0.018505, 0.043283, -0.000125, -0.000000, 3.141593, -0.000000]),accel_mss,speed_ms,0,0.001)
    |   movel(pose_trans(ref_frame,p[0.019275, 0.044186, -0.000125, -0.000000, 3.141593, 0.000000]),accel_mss,speed_ms,0,0.001)
    |   movel(pose_trans(ref_frame,p[0.020122, 0.045016, -0.000125, -0.000000, 3.141593, 0.000000]),accel_mss,speed_ms,0,0.001)
    |   movel(pose_trans(ref_frame,p[0.020969, 0.045613, -0.000125, 0.000000, 3.141593, -0.000000]),accel_mss,speed_ms,0,0.001)
    |   movel(pose_trans(ref_frame,p[0.021769, 0.046216, -0.000125, -0.000000, 3.141593, -0.000000]),accel_mss,speed_ms,0,0.001)
    |   movel(pose_trans(ref_frame,p[0.022826, 0.048008, -0.000125, 0.000000, 3.141593, 0.000000]),accel_mss,speed_ms,0,0.001)
    |   movel(pose_trans(ref_frame,p[0.023320, 0.050014, -0.000125, -0.000000, 3.141593, 0.000000]),accel_mss,speed_ms,0,0) # end trace
    |   speed_ms    = 1.000
    |   movel(pose_trans(ref_frame,p[0.023320, 0.050014, 0.005000, -0.000000, 3.141593, 0.000000]),accel_mss,speed_ms,0,0.001)
    |   movel(pose_trans(ref_frame,p[0.015765, 0.045388, 0.005000, 0.000000, 3.141593, 0.000000]),accel_mss,speed_ms,0,0) # end trace
    |   speed_ms    = 0.002
    |   movel(pose_trans(ref_frame,p[0.015765, 0.045388, -0.000125, 0.000000, 3.141593, -0.000000]),accel_mss,speed_ms,0,0) # end trace
    |   speed_ms    = 0.007
    |   movel(pose_trans(ref_frame,p[0.015496, 0.045683, -0.000125, 0.000000, 3.141593, 0.000000]),accel_mss,speed_ms,0,0.001)
    |   movel(pose_trans(ref_frame,p[0.015721, 0.046101, -0.000125, -0.000000, 3.141593, -0.000000]),accel_mss,speed_ms,0,0.001)
    |   movel(pose_trans(ref_frame,p[0.016157, 0.046234, -0.000125, -0.000000, 3.141593, -0.000000]),accel_mss,speed_ms,0,0.001)
    |   movel(pose_trans(ref_frame,p[0.016630, 0.046258, -0.000125, -0.000000, 3.141593, 0.000000]),accel_mss,speed_ms,0,0.001)
    |   movel(pose_trans(ref_frame,p[0.017863, 0.046761, -0.000125, 0.000000, 3.141593, -0.000000]),accel_mss,speed_ms,0,0.001)
    |   movel(pose_trans(ref_frame,p[0.018882, 0.047707, -0.000125, 0.000000, 3.141593, 0.000000]),accel_mss,speed_ms,0,0.001)
    |   movel(pose_trans(ref_frame,p[0.018989, 0.047837, -0.000125, -0.000000, 3.141593, -0.000000]),accel_mss,speed_ms,0,0.001)
    |   movel(pose_trans(ref_frame,p[0.019035, 0.047990, -0.000125, -0.000000, 3.141593, -0.000000]),accel_mss,speed_ms,0,0.001)
    |   movel(pose_trans(ref_frame,p[0.018959, 0.048158, -0.000125, 0.000000, 3.141593, -0.000000]),accel_mss,speed_ms,0,0.001)
    |   movel(pose_trans(ref_frame,p[0.018795, 0.048276, -0.000125, 0.000000, 3.141593, 0.000000]),accel_mss,speed_ms,0,0.001)
    |   movel(pose_trans(ref_frame,p[0.017095, 0.048692, -0.000125, 0.000000, 3.141593, 0.000000]),accel_mss,speed_ms,0,0.001)
    |   movel(pose_trans(ref_frame,p[0.015433, 0.048144, -0.000125, -0.000000, 3.141593, -0.000000]),accel_mss,speed_ms,0,0.001)
    |   movel(pose_trans(ref_frame,p[0.015341, 0.048635, -0.000125, -0.000000, 3.141593, -0.000000]),accel_mss,speed_ms,0,0.001)
    |   movel(pose_trans(ref_frame,p[0.014909, 0.048937, -0.000125, 0.000000, 3.141593, 0.000000]),accel_mss,speed_ms,0,0.001)
    |   movel(pose_trans(ref_frame,p[0.014393, 0.048959, -0.000125, 0.000000, 3.141593, 0.000000]),accel_mss,speed_ms,0,0.001)
    |   movel(pose_trans(ref_frame,p[0.013887, 0.048800, -0.000125, -0.000000, 3.141593, -0.000000]),accel_mss,speed_ms,0,0.001)
    |   movel(pose_trans(ref_frame,p[0.012757, 0.048059, -0.000125, -0.000000, 3.141593, -0.000000]),accel_mss,speed_ms,0,0.001)
    |   movel(pose_trans(ref_frame,p[0.011943, 0.046981, -0.000125, 0.000000, 3.141593, -0.000000]),accel_mss,speed_ms,0,0.001)
    |   movel(pose_trans(ref_frame,p[0.011857, 0.046770, -0.000125, 0.000000, 3.141593, -0.000000]),accel_mss,speed_ms,0,0.001)
    |   movel(pose_trans(ref_frame,p[0.011855, 0.046551, -0.000125, -0.000000, 3.141593, -0.000000]),accel_mss,speed_ms,0,0.001)
    |   movel(pose_trans(ref_frame,p[0.011948, 0.046392, -0.000125, 0.000000, 3.141593, -0.000000]),accel_mss,speed_ms,0,0.001)
    |   movel(pose_trans(ref_frame,p[0.012091, 0.046267, -0.000125, -0.000000, 3.141593, 0.000000]),accel_mss,speed_ms,0,0.001)
    |   movel(pose_trans(ref_frame,p[0.013146, 0.045670, -0.000125, -0.000000, 3.141593, 0.000000]),accel_mss,speed_ms,0,0.001)
    |   movel(pose_trans(ref_frame,p[0.014158, 0.044991, -0.000125, 0.000000, 3.141593, 0.000000]),accel_mss,speed_ms,0,0.001)
    |   movel(pose_trans(ref_frame,p[0.013569, 0.044459, -0.000125, -0.000000, 3.141593, -0.000000]),accel_mss,speed_ms,0,0.001)
    |   movel(pose_trans(ref_frame,p[0.012858, 0.044132, -0.000125, 0.000000, 3.141593, -0.000000]),accel_mss,speed_ms,0,0.001)
    |   movel(pose_trans(ref_frame,p[0.012299, 0.044094, -0.000125, -0.000000, 3.141593, 0.000000]),accel_mss,speed_ms,0,0.001)
    |   movel(pose_trans(ref_frame,p[0.011761, 0.044224, -0.000125, -0.000000, 3.141593, -0.000000]),accel_mss,speed_ms,0,0.001)
    |   movel(pose_trans(ref_frame,p[0.011444, 0.044435, -0.000125, -0.000000, 3.141593, -0.000000]),accel_mss,speed_ms,0,0.001)
    |   movel(pose_trans(ref_frame,p[0.011278, 0.044765, -0.000125, 0.000000, 3.141593, 0.000000]),accel_mss,speed_ms,0,0.001)
    |   movel(pose_trans(ref_frame,p[0.011385, 0.045225, -0.000125, -0.000000, 3.141593, -0.000000]),accel_mss,speed_ms,0,0.001)
    |   movel(pose_trans(ref_frame,p[0.011724, 0.045598, -0.000125, -0.000000, 3.141593, -0.000000]),accel_mss,speed_ms,0,0) # end trace
    |   speed_ms    = 1.000
    |   movel(pose_trans(ref_frame,p[0.011724, 0.045598, 0.005000, -0.000000, 3.141593, 0.000000]),accel_mss,speed_ms,0,0.001)
    |   movel(pose_trans(ref_frame,p[0.011374, 0.047442, 0.005000, -0.000000, 3.141593, -0.000000]),accel_mss,speed_ms,0,0) # end trace
    |   speed_ms    = 0.002
    |   movel(pose_trans(ref_frame,p[0.011374, 0.047442, -0.000125, -0.000000, 3.141593, -0.000000]),accel_mss,speed_ms,0,0) # end trace
    |   speed_ms    = 0.007
    |   movel(pose_trans(ref_frame,p[0.010402, 0.046839, -0.000125, -0.000000, 3.141593, -0.000000]),accel_mss,speed_ms,0,0.001)
    |   movel(pose_trans(ref_frame,p[0.009754, 0.045820, -0.000125, -0.000000, 3.141593, 0.000000]),accel_mss,speed_ms,0,0.001)
    |   movel(pose_trans(ref_frame,p[0.008506, 0.042222, -0.000125, -0.000000, 3.141593, -0.000000]),accel_mss,speed_ms,0,0.001)
    |   movel(pose_trans(ref_frame,p[0.008199, 0.038426, -0.000125, -0.000000, 3.141593, -0.000000]),accel_mss,speed_ms,0,0.001)
    |   movel(pose_trans(ref_frame,p[0.008272, 0.037764, -0.000125, 0.000000, 3.141593, -0.000000]),accel_mss,speed_ms,0,0.001)
    |   movel(pose_trans(ref_frame,p[0.008531, 0.037168, -0.000125, -0.000000, 3.141593, 0.000000]),accel_mss,speed_ms,0,0.001)
    |   movel(pose_trans(ref_frame,p[0.009078, 0.036670, -0.000125, 0.000000, 3.141593, -0.000000]),accel_mss,speed_ms,0,0.001)
    |   movel(pose_trans(ref_frame,p[0.009569, 0.036139, -0.000125, -0.000000, 3.141593, -0.000000]),accel_mss,speed_ms,0,0.001)
    |   movel(pose_trans(ref_frame,p[0.009661, 0.035352, -0.000125, -0.000000, 3.141593, -0.000000]),accel_mss,speed_ms,0,0.001)
    |   movel(pose_trans(ref_frame,p[0.009438, 0.034539, -0.000125, 0.000000, 3.141593, -0.000000]),accel_mss,speed_ms,0,0.001)
    |   movel(pose_trans(ref_frame,p[0.009130, 0.032795, -0.000125, 0.000000, 3.141593, -0.000000]),accel_mss,speed_ms,0,0.001)
    |   movel(pose_trans(ref_frame,p[0.009256, 0.031028, -0.000125, -0.000000, 3.141593, 0.000000]),accel_mss,speed_ms,0,0.001)
    |   movel(pose_trans(ref_frame,p[0.009606, 0.029909, -0.000125, 0.000000, 3.141593, -0.000000]),accel_mss,speed_ms,0,0.001)
    |   movel(pose_trans(ref_frame,p[0.010279, 0.028973, -0.000125, -0.000000, 3.141593, -0.000000]),accel_mss,speed_ms,0,0.001)
    |   movel(pose_trans(ref_frame,p[0.011322, 0.028449, -0.000125, -0.000000, 3.141593, -0.000000]),accel_mss,speed_ms,0,0.001)
    |   movel(pose_trans(ref_frame,p[0.012435, 0.028644, -0.000125, -0.000000, 3.141593, -0.000000]),accel_mss,speed_ms,0,0) # end trace
    |   speed_ms    = 1.000
    |   movel(pose_trans(ref_frame,p[0.012435, 0.028644, 0.005000, -0.000000, 3.141593, -0.000000]),accel_mss,speed_ms,0,0.001)
    |   movel(pose_trans(ref_frame,p[0.040152, 0.062572, 0.005000, -0.000000, 3.141593, 0.000000]),accel_mss,speed_ms,0,0) # end trace
    |   speed_ms    = 0.002
    |   movel(pose_trans(ref_frame,p[0.040152, 0.062572, -0.000125, -0.000000, 3.141593, 0.000000]),accel_mss,speed_ms,0,0) # end trace
    |   speed_ms    = 0.007
    |   movel(pose_trans(ref_frame,p[0.041280, 0.061304, -0.000125, -0.000000, 3.141593, 0.000000]),accel_mss,speed_ms,0,0.001)
    |   movel(pose_trans(ref_frame,p[0.041904, 0.059657, -0.000125, -0.000000, 3.141593, 0.000000]),accel_mss,speed_ms,0,0.001)
    |   movel(pose_trans(ref_frame,p[0.043428, 0.050774, -0.000125, 0.000000, 3.141593, 0.000000]),accel_mss,speed_ms,0,0.001)
    |   movel(pose_trans(ref_frame,p[0.043651, 0.041780, -0.000125, 0.000000, 3.141593, -0.000000]),accel_mss,speed_ms,0,0.001)
    |   movel(pose_trans(ref_frame,p[0.043440, 0.032724, -0.000125, 0.000000, 3.141593, -0.000000]),accel_mss,speed_ms,0,0.001)
    |   movel(pose_trans(ref_frame,p[0.043840, 0.023683, -0.000125, 0.000000, 3.141593, -0.000000]),accel_mss,speed_ms,0,0.001)
    |   movel(pose_trans(ref_frame,p[0.044186, 0.021637, -0.000125, 0.000000, 3.141593, -0.000000]),accel_mss,speed_ms,0,0.001)
    |   movel(pose_trans(ref_frame,p[0.044782, 0.019655, -0.000125, -0.000000, 3.141593, -0.000000]),accel_mss,speed_ms,0,0.001)
    |   movel(pose_trans(ref_frame,p[0.049207, 0.015182, -0.000125, -0.000000, 3.141593, -0.000000]),accel_mss,speed_ms,0,0.001)
    |   movel(pose_trans(ref_frame,p[0.055498, 0.014807, -0.000125, 0.000000, 3.141593, -0.000000]),accel_mss,speed_ms,0,0.001)
    |   movel(pose_trans(ref_frame,p[0.058841, 0.016792, -0.000125, 0.000000, 3.141593, 0.000000]),accel_mss,speed_ms,0,0.001)
    |   movel(pose_trans(ref_frame,p[0.060627, 0.020253, -0.000125, -0.000000, 3.141593, -0.000000]),accel_mss,speed_ms,0,0.001)
    |   movel(pose_trans(ref_frame,p[0.060755, 0.022937, -0.000125, 0.000000, 3.141593, -0.000000]),accel_mss,speed_ms,0,0.001)
    |   movel(pose_trans(ref_frame,p[0.060329, 0.025608, -0.000125, -0.000000, 3.141593, -0.000000]),accel_mss,speed_ms,0,0.001)
    |   movel(pose_trans(ref_frame,p[0.059618, 0.027570, -0.000125, 0.000000, 3.141593, 0.000000]),accel_mss,speed_ms,0,0.001)
    |   movel(pose_trans(ref_frame,p[0.058741, 0.029477, -0.000125, 0.000000, 3.141593, -0.000000]),accel_mss,speed_ms,0,0.001)
    |   movel(pose_trans(ref_frame,p[0.058073, 0.032154, -0.000125, -0.000000, 3.141593, -0.000000]),accel_mss,speed_ms,0,0.001)
    |   movel(pose_trans(ref_frame,p[0.058370, 0.034935, -0.000125, -0.000000, 3.141593, 0.000000]),accel_mss,speed_ms,0,0) # end trace
    |   speed_ms    = 1.000
    |   movel(pose_trans(ref_frame,p[0.058370, 0.034935, 0.005000, -0.000000, 3.141593, 0.000000]),accel_mss,speed_ms,0,0.001)
    |   movel(pose_trans(ref_frame,p[0.058811, 0.068348, 0.005000, -0.000000, 3.141593, 0.000000]),accel_mss,speed_ms,0,0) # end trace
    |   speed_ms    = 0.002
    |   movel(pose_trans(ref_frame,p[0.058811, 0.068348, -0.000125, -0.000000, 3.141593, -0.000000]),accel_mss,speed_ms,0,0) # end trace
    |   speed_ms    = 0.007
    |   movel(pose_trans(ref_frame,p[0.060233, 0.071971, -0.000125, 0.000000, 3.141593, -0.000000]),accel_mss,speed_ms,0,0.001)
    |   movel(pose_trans(ref_frame,p[0.062473, 0.075171, -0.000125, 0.000000, 3.141593, 0.000000]),accel_mss,speed_ms,0,0.001)
    |   movel(pose_trans(ref_frame,p[0.061941, 0.074365, -0.000125, 0.000000, 3.141593, 0.000000]),accel_mss,speed_ms,0,0.001)
    |   movel(pose_trans(ref_frame,p[0.061985, 0.073384, -0.000125, -0.000000, 3.141593, -0.000000]),accel_mss,speed_ms,0,0.001)
    |   movel(pose_trans(ref_frame,p[0.063874, 0.073596, -0.000125, 0.000000, 3.141593, 0.000000]),accel_mss,speed_ms,0,0.001)
    |   movel(pose_trans(ref_frame,p[0.065099, 0.076066, -0.000125, 0.000000, 3.141593, -0.000000]),accel_mss,speed_ms,0,0.001)
    |   movel(pose_trans(ref_frame,p[0.065959, 0.077076, -0.000125, -0.000000, 3.141593, 0.000000]),accel_mss,speed_ms,0,0.001)
    |   movel(pose_trans(ref_frame,p[0.066998, 0.077868, -0.000125, 0.000000, 3.141593, 0.000000]),accel_mss,speed_ms,0,0.001)
    |   movel(pose_trans(ref_frame,p[0.066447, 0.076772, -0.000125, 0.000000, 3.141593, -0.000000]),accel_mss,speed_ms,0,0.001)
    |   movel(pose_trans(ref_frame,p[0.067033, 0.075482, -0.000125, -0.000000, 3.141593, 0.000000]),accel_mss,speed_ms,0,0.001)
    |   movel(pose_trans(ref_frame,p[0.068043, 0.075397, -0.000125, 0.000000, 3.141593, 0.000000]),accel_mss,speed_ms,0,0.001)
    |   movel(pose_trans(ref_frame,p[0.068731, 0.075995, -0.000125, -0.000000, 3.141593, -0.000000]),accel_mss,speed_ms,0,0.001)
    |   movel(pose_trans(ref_frame,p[0.069987, 0.076897, -0.000125, -0.000000, 3.141593, 0.000000]),accel_mss,speed_ms,0,0.001)
    |   movel(pose_trans(ref_frame,p[0.071493, 0.077367, -0.000125, -0.000000, 3.141593, 0.000000]),accel_mss,speed_ms,0,0.001)
    |   movel(pose_trans(ref_frame,p[0.071058, 0.076946, -0.000125, 0.000000, 3.141593, -0.000000]),accel_mss,speed_ms,0,0.001)
    |   movel(pose_trans(ref_frame,p[0.070714, 0.076456, -0.000125, 0.000000, 3.141593, 0.000000]),accel_mss,speed_ms,0,0.001)
    |   movel(pose_trans(ref_frame,p[0.070576, 0.075867, -0.000125, 0.000000, 3.141593, 0.000000]),accel_mss,speed_ms,0,0.001)
    |   movel(pose_trans(ref_frame,p[0.070770, 0.075316, -0.000125, -0.000000, 3.141593, -0.000000]),accel_mss,speed_ms,0,0.001)
    |   movel(pose_trans(ref_frame,p[0.071417, 0.074970, -0.000125, 0.000000, 3.141593, 0.000000]),accel_mss,speed_ms,0,0.001)
    |   movel(pose_trans(ref_frame,p[0.072209, 0.074970, -0.000125, 0.000000, 3.141593, -0.000000]),accel_mss,speed_ms,0,0) # end trace
    |   speed_ms    = 1.000
    |   movel(pose_trans(ref_frame,p[0.072209, 0.074970, 0.005000, 0.000000, 3.141593, -0.000000]),accel_mss,speed_ms,0,0.001)
    |   movel(pose_trans(ref_frame,p[0.000000, 0.000000, 0.005000, 0.000000, 3.141593, -0.000000]),accel_mss,speed_ms,0,0.001)
    |   movel(pose_trans(ref_frame,p[0.000000, 0.000000, 0.105000, 0.000000, 3.141593, -0.000000]),accel_mss,speed_ms,0,0.001)
    |   # End of main program
    | end
    | 
    | azat_dragon_rotate()
  Halt
